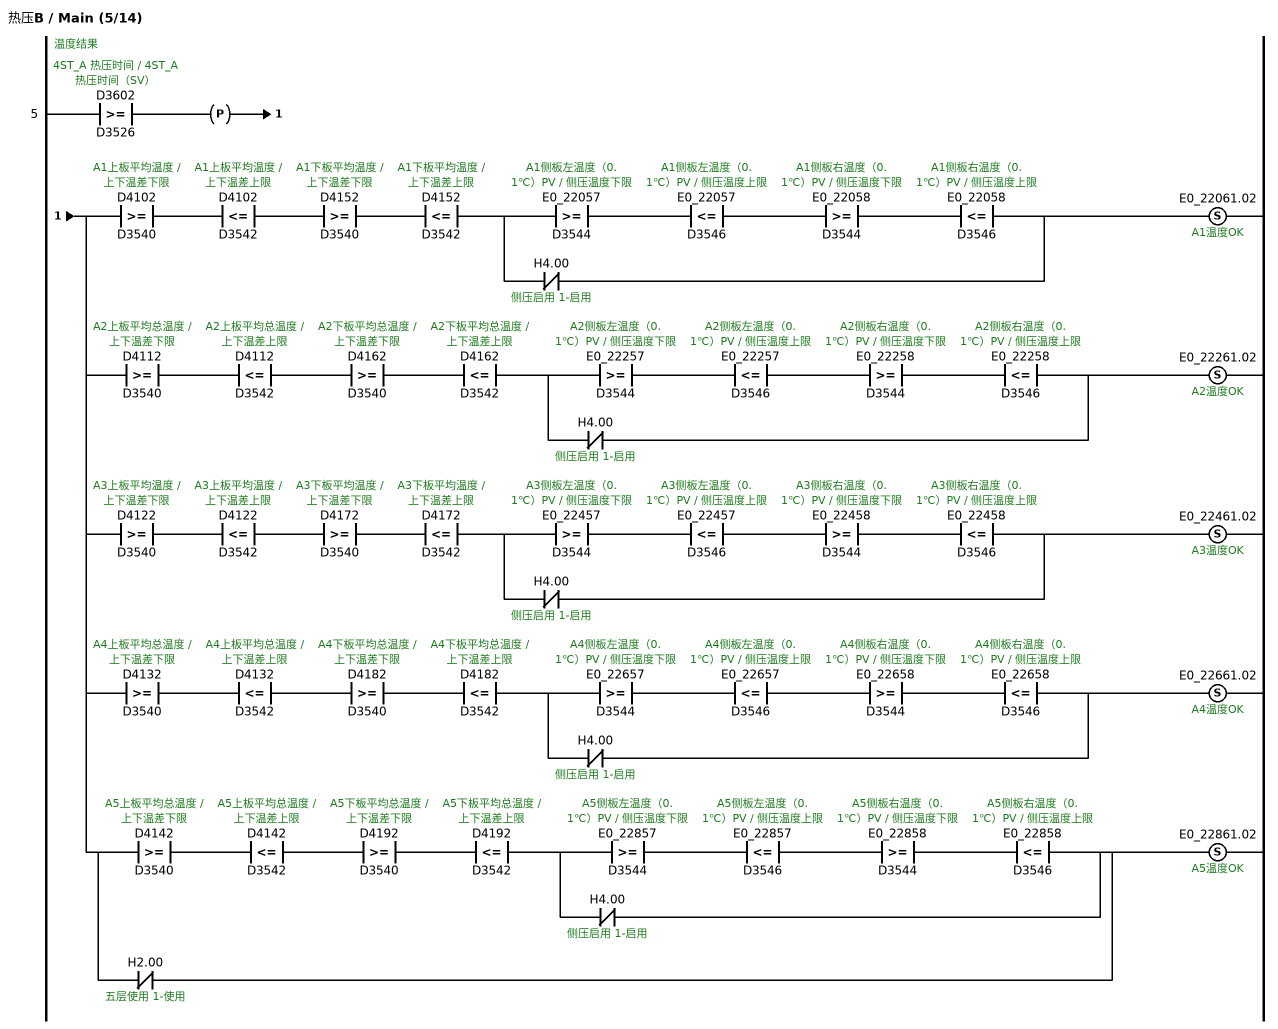
; [picture p168: 热压B / Main, rungs 5-5]
; rung 5: 温度结果
LD>=(325) D3602 D3526  ; 4ST_A 热压时间, 4ST_A 热压时间（SV）
UP(521)
OUT TR0
AND>=(325) D4102 D3540  ; A1上板平均温度, 上下温差下限
AND<=(315) D4102 D3542  ; A1上板平均温度, 上下温差上限
AND>=(325) D4152 D3540  ; A1下板平均温度, 上下温差下限
AND<=(315) D4152 D3542  ; A1下板平均温度, 上下温差上限
LD>=(325) E0_22057 D3544  ; A1侧板左温度（0.1℃）PV, 侧压温度下限
AND<=(315) E0_22057 D3546  ; A1侧板左温度（0.1℃）PV, 侧压温度上限
AND>=(325) E0_22058 D3544  ; A1侧板右温度（0.1℃）PV, 侧压温度下限
AND<=(315) E0_22058 D3546  ; A1侧板右温度（0.1℃）PV, 侧压温度上限
ORNOT H4.00  ; 侧压启用 1-启用
ANDLD
SET E0_22061.02  ; A1温度OK
LD TR0
AND>=(325) D4112 D3540  ; A2上板平均总温度, 上下温差下限
AND<=(315) D4112 D3542  ; A2上板平均总温度, 上下温差上限
AND>=(325) D4162 D3540  ; A2下板平均总温度, 上下温差下限
AND<=(315) D4162 D3542  ; A2下板平均总温度, 上下温差上限
LD>=(325) E0_22257 D3544  ; A2侧板左温度（0.1℃）PV, 侧压温度下限
AND<=(315) E0_22257 D3546  ; A2侧板左温度（0.1℃）PV, 侧压温度上限
AND>=(325) E0_22258 D3544  ; A2侧板右温度（0.1℃）PV, 侧压温度下限
AND<=(315) E0_22258 D3546  ; A2侧板右温度（0.1℃）PV, 侧压温度上限
ORNOT H4.00  ; 侧压启用 1-启用
ANDLD
SET E0_22261.02  ; A2温度OK
LD TR0
AND>=(325) D4122 D3540  ; A3上板平均温度, 上下温差下限
AND<=(315) D4122 D3542  ; A3上板平均温度, 上下温差上限
AND>=(325) D4172 D3540  ; A3下板平均温度, 上下温差下限
AND<=(315) D4172 D3542  ; A3下板平均温度, 上下温差上限
LD>=(325) E0_22457 D3544  ; A3侧板左温度（0.1℃）PV, 侧压温度下限
AND<=(315) E0_22457 D3546  ; A3侧板左温度（0.1℃）PV, 侧压温度上限
AND>=(325) E0_22458 D3544  ; A3侧板右温度（0.1℃）PV, 侧压温度下限
AND<=(315) E0_22458 D3546  ; A3侧板右温度（0.1℃）PV, 侧压温度上限
ORNOT H4.00  ; 侧压启用 1-启用
ANDLD
SET E0_22461.02  ; A3温度OK
LD TR0
AND>=(325) D4132 D3540  ; A4上板平均总温度, 上下温差下限
AND<=(315) D4132 D3542  ; A4上板平均总温度, 上下温差上限
AND>=(325) D4182 D3540  ; A4下板平均总温度, 上下温差下限
AND<=(315) D4182 D3542  ; A4下板平均总温度, 上下温差上限
LD>=(325) E0_22657 D3544  ; A4侧板左温度（0.1℃）PV, 侧压温度下限
AND<=(315) E0_22657 D3546  ; A4侧板左温度（0.1℃）PV, 侧压温度上限
AND>=(325) E0_22658 D3544  ; A4侧板右温度（0.1℃）PV, 侧压温度下限
AND<=(315) E0_22658 D3546  ; A4侧板右温度（0.1℃）PV, 侧压温度上限
ORNOT H4.00  ; 侧压启用 1-启用
ANDLD
SET E0_22661.02  ; A4温度OK
LD TR0
LD>=(325) D4142 D3540  ; A5上板平均总温度, 上下温差下限
AND<=(315) D4142 D3542  ; A5上板平均总温度, 上下温差上限
AND>=(325) D4192 D3540  ; A5下板平均总温度, 上下温差下限
AND<=(315) D4192 D3542  ; A5下板平均总温度, 上下温差上限
LD>=(325) E0_22857 D3544  ; A5侧板左温度（0.1℃）PV, 侧压温度下限
AND<=(315) E0_22857 D3546  ; A5侧板左温度（0.1℃）PV, 侧压温度上限
AND>=(325) E0_22858 D3544  ; A5侧板右温度（0.1℃）PV, 侧压温度下限
AND<=(315) E0_22858 D3546  ; A5侧板右温度（0.1℃）PV, 侧压温度上限
ORNOT H4.00  ; 侧压启用 1-启用
ANDLD
ORNOT H2.00  ; 五层使用 1-使用
ANDLD
SET E0_22861.02  ; A5温度OK

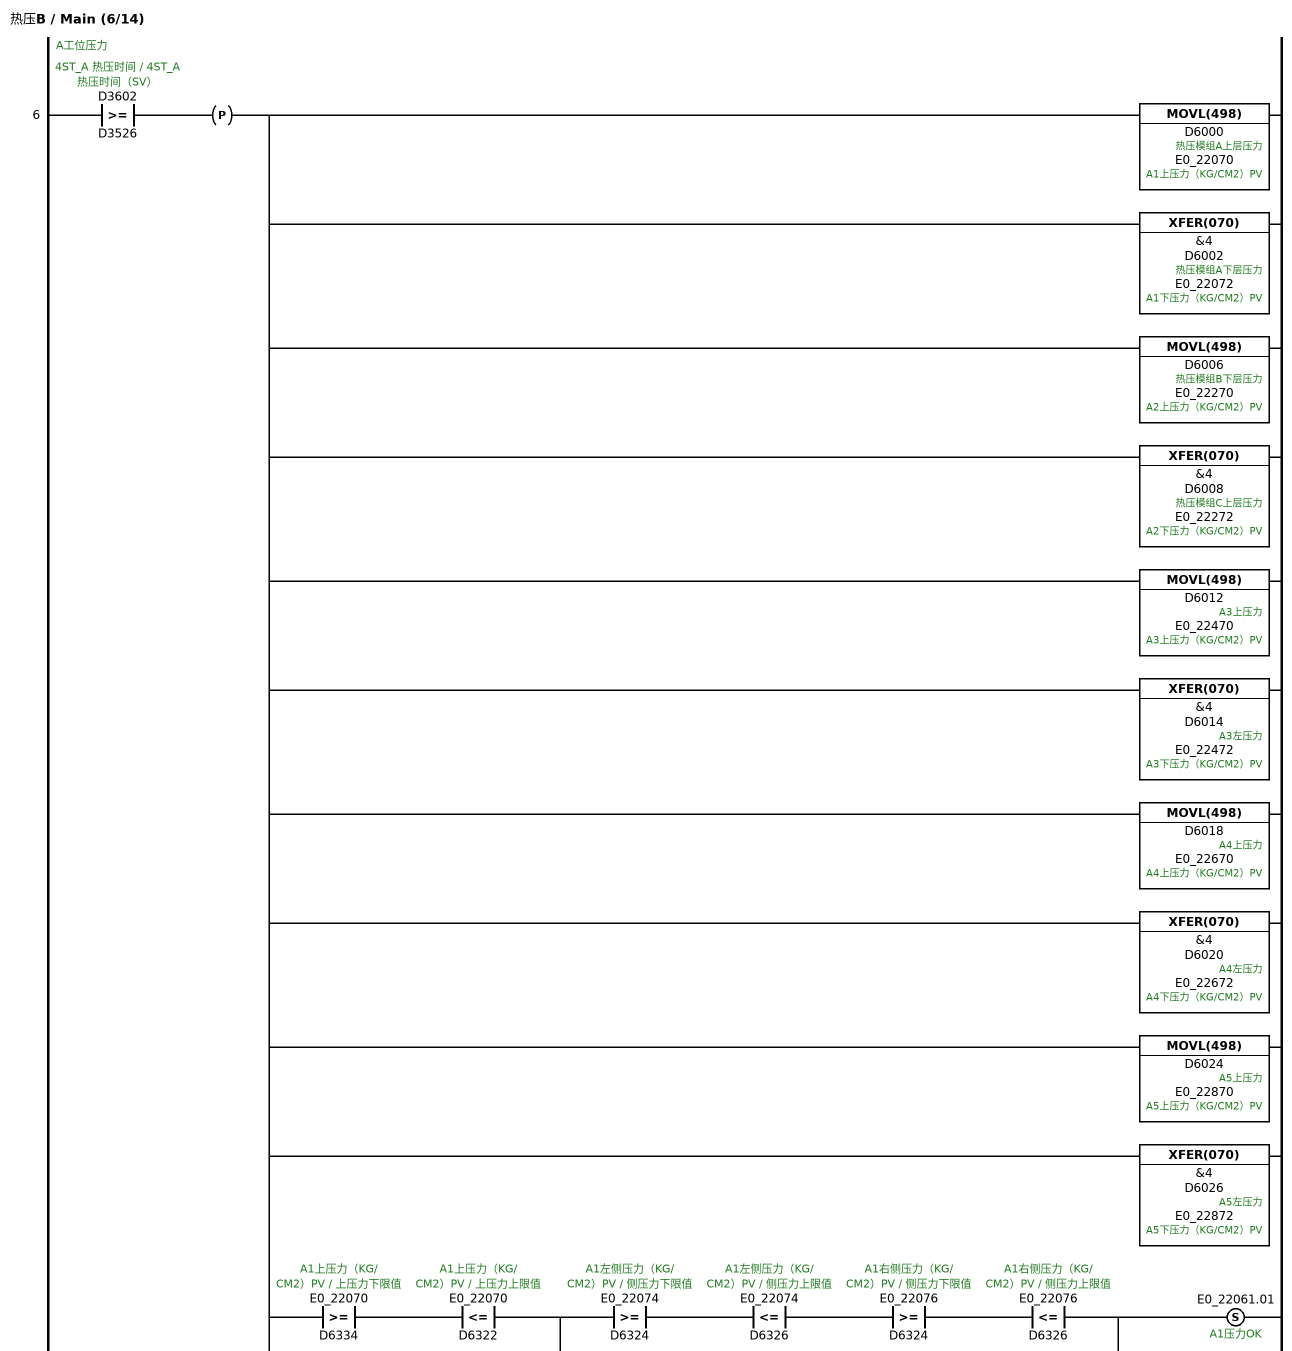

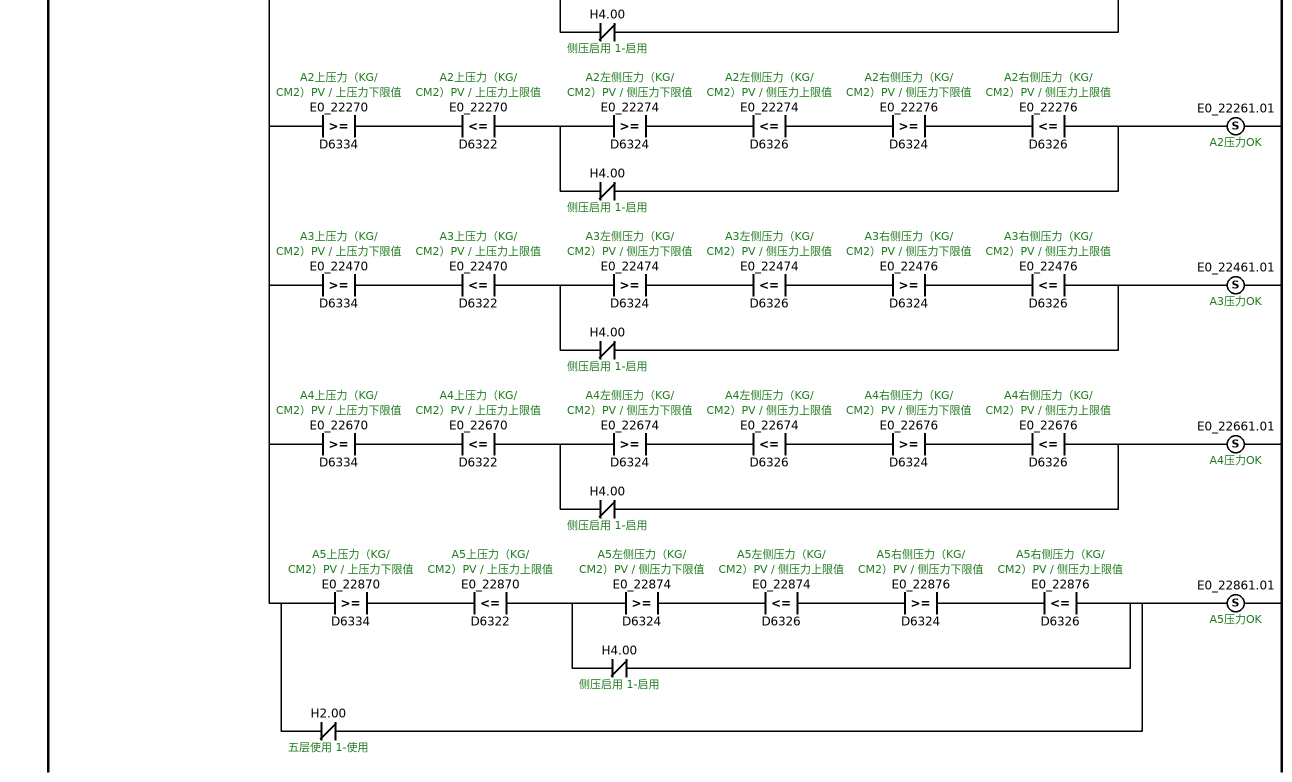
; rung 6: A工位压力
LD>=(325) D3602 D3526  ; 4ST_A 热压时间, 4ST_A 热压时间（SV）
UP(521)
OUT TR0
MOVL(498) D6000 E0_22070  ; 热压模组A上层压力, A1上压力（KG/CM2）PV
XFER(070) &4 D6002 E0_22072  ; 热压模组A下层压力, A1下压力（KG/CM2）PV
MOVL(498) D6006 E0_22270  ; 热压模组B下层压力, A2上压力（KG/CM2）PV
XFER(070) &4 D6008 E0_22272  ; 热压模组C上层压力, A2下压力（KG/CM2）PV
MOVL(498) D6012 E0_22470  ; A3上压力, A3上压力（KG/CM2）PV
XFER(070) &4 D6014 E0_22472  ; A3左压力, A3下压力（KG/CM2）PV
MOVL(498) D6018 E0_22670  ; A4上压力, A4上压力（KG/CM2）PV
XFER(070) &4 D6020 E0_22672  ; A4左压力, A4下压力（KG/CM2）PV
MOVL(498) D6024 E0_22870  ; A5上压力, A5上压力（KG/CM2）PV
XFER(070) &4 D6026 E0_22872  ; A5左压力, A5下压力（KG/CM2）PV
AND>=L(326) E0_22070 D6334  ; A1上压力（KG/CM2）PV, 上压力下限值
AND<=L(316) E0_22070 D6322  ; A1上压力（KG/CM2）PV, 上压力上限值
LD>=L(326) E0_22074 D6324  ; A1左侧压力（KG/CM2）PV, 侧压力下限值
AND<=L(316) E0_22074 D6326  ; A1左侧压力（KG/CM2）PV, 侧压力上限值
AND>=L(326) E0_22076 D6324  ; A1右侧压力（KG/CM2）PV, 侧压力下限值
AND<=L(316) E0_22076 D6326  ; A1右侧压力（KG/CM2）PV, 侧压力上限值
ORNOT H4.00  ; 侧压启用 1-启用
ANDLD
SET E0_22061.01  ; A1压力OK
LD TR0
AND>=L(326) E0_22270 D6334  ; A2上压力（KG/CM2）PV, 上压力下限值
AND<=L(316) E0_22270 D6322  ; A2上压力（KG/CM2）PV, 上压力上限值
LD>=L(326) E0_22274 D6324  ; A2左侧压力（KG/CM2）PV, 侧压力下限值
AND<=L(316) E0_22274 D6326  ; A2左侧压力（KG/CM2）PV, 侧压力上限值
AND>=L(326) E0_22276 D6324  ; A2右侧压力（KG/CM2）PV, 侧压力下限值
AND<=L(316) E0_22276 D6326  ; A2右侧压力（KG/CM2）PV, 侧压力上限值
ORNOT H4.00  ; 侧压启用 1-启用
ANDLD
SET E0_22261.01  ; A2压力OK
LD TR0
AND>=L(326) E0_22470 D6334  ; A3上压力（KG/CM2）PV, 上压力下限值
AND<=L(316) E0_22470 D6322  ; A3上压力（KG/CM2）PV, 上压力上限值
LD>=L(326) E0_22474 D6324  ; A3左侧压力（KG/CM2）PV, 侧压力下限值
AND<=L(316) E0_22474 D6326  ; A3左侧压力（KG/CM2）PV, 侧压力上限值
AND>=L(326) E0_22476 D6324  ; A3右侧压力（KG/CM2）PV, 侧压力下限值
AND<=L(316) E0_22476 D6326  ; A3右侧压力（KG/CM2）PV, 侧压力上限值
ORNOT H4.00  ; 侧压启用 1-启用
ANDLD
SET E0_22461.01  ; A3压力OK
LD TR0
AND>=L(326) E0_22670 D6334  ; A4上压力（KG/CM2）PV, 上压力下限值
AND<=L(316) E0_22670 D6322  ; A4上压力（KG/CM2）PV, 上压力上限值
LD>=L(326) E0_22674 D6324  ; A4左侧压力（KG/CM2）PV, 侧压力下限值
AND<=L(316) E0_22674 D6326  ; A4左侧压力（KG/CM2）PV, 侧压力上限值
AND>=L(326) E0_22676 D6324  ; A4右侧压力（KG/CM2）PV, 侧压力下限值
AND<=L(316) E0_22676 D6326  ; A4右侧压力（KG/CM2）PV, 侧压力上限值
ORNOT H4.00  ; 侧压启用 1-启用
ANDLD
SET E0_22661.01  ; A4压力OK
LD TR0
LD>=L(326) E0_22870 D6334  ; A5上压力（KG/CM2）PV, 上压力下限值
AND<=L(316) E0_22870 D6322  ; A5上压力（KG/CM2）PV, 上压力上限值
LD>=L(326) E0_22874 D6324  ; A5左侧压力（KG/CM2）PV, 侧压力下限值
AND<=L(316) E0_22874 D6326  ; A5左侧压力（KG/CM2）PV, 侧压力上限值
AND>=L(326) E0_22876 D6324  ; A5右侧压力（KG/CM2）PV, 侧压力下限值
AND<=L(316) E0_22876 D6326  ; A5右侧压力（KG/CM2）PV, 侧压力上限值
ORNOT H4.00  ; 侧压启用 1-启用
ANDLD
ORNOT H2.00  ; 五层使用 1-使用
ANDLD
SET E0_22861.01  ; A5压力OK

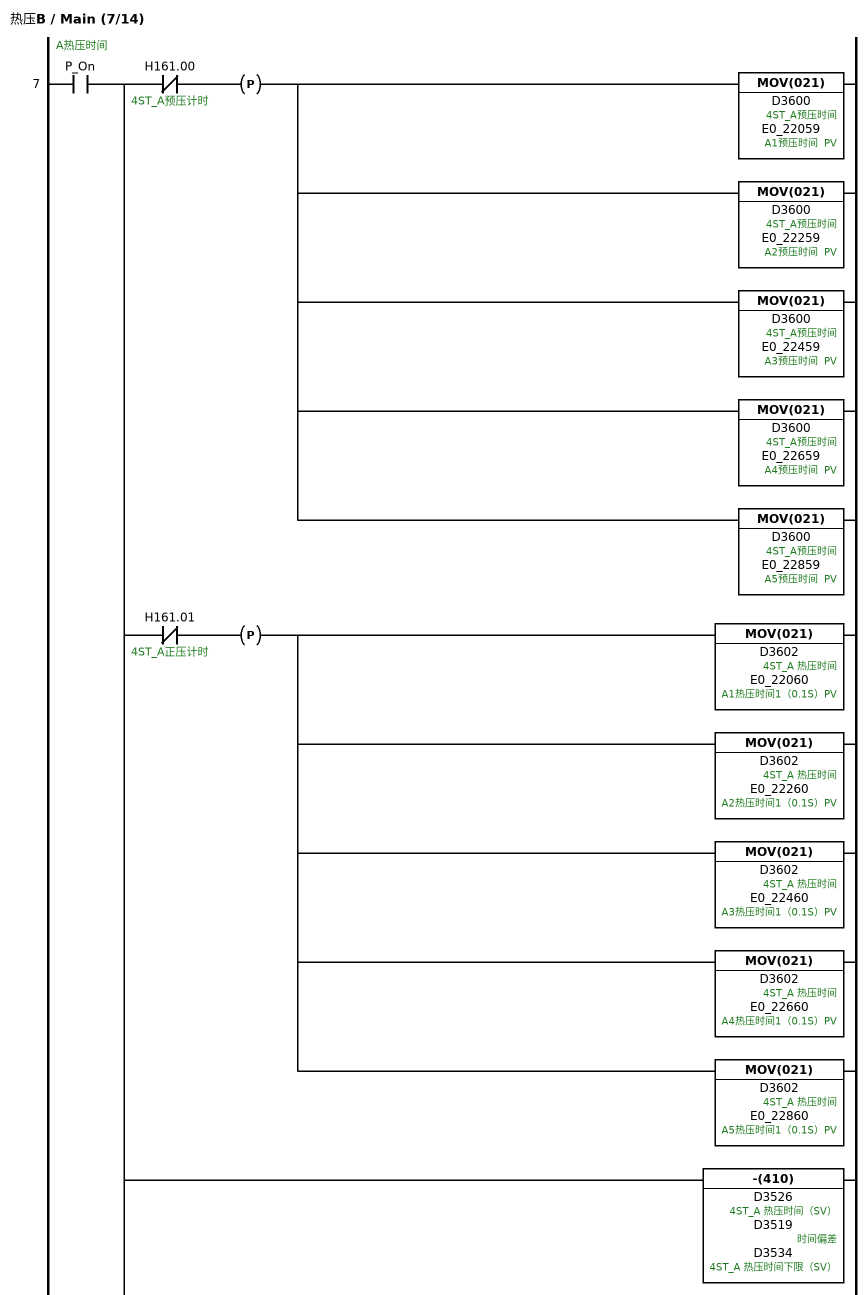

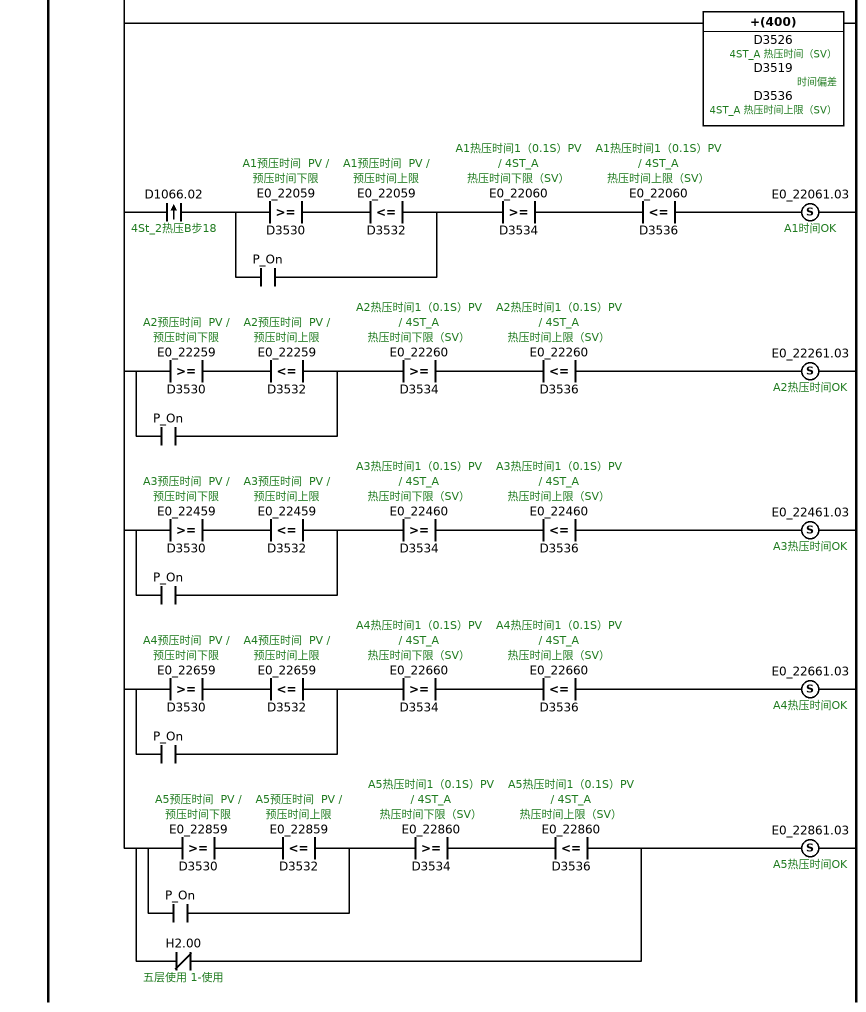
; rung 7: A热压时间
LD P_On
OUT TR0
ANDNOT H161.00  ; 4ST_A预压计时
UP(521)
MOV(021) D3600 E0_22059  ; 4ST_A预压时间, A1预压时间  PV
MOV(021) D3600 E0_22259  ; 4ST_A预压时间, A2预压时间  PV
MOV(021) D3600 E0_22459  ; 4ST_A预压时间, A3预压时间  PV
MOV(021) D3600 E0_22659  ; 4ST_A预压时间, A4预压时间  PV
MOV(021) D3600 E0_22859  ; 4ST_A预压时间, A5预压时间  PV
LD TR0
ANDNOT H161.01  ; 4ST_A正压计时
UP(521)
MOV(021) D3602 E0_22060  ; 4ST_A 热压时间, A1热压时间1（0.1S）PV
MOV(021) D3602 E0_22260  ; 4ST_A 热压时间, A2热压时间1（0.1S）PV
MOV(021) D3602 E0_22460  ; 4ST_A 热压时间, A3热压时间1（0.1S）PV
MOV(021) D3602 E0_22660  ; 4ST_A 热压时间, A4热压时间1（0.1S）PV
MOV(021) D3602 E0_22860  ; 4ST_A 热压时间, A5热压时间1（0.1S）PV
LD TR0
-(410) D3526 D3519 D3534  ; 4ST_A 热压时间（SV）, 时间偏差, 4ST_A 热压时间下限（SV）
+(400) D3526 D3519 D3536  ; 4ST_A 热压时间（SV）, 时间偏差, 4ST_A 热压时间上限（SV）
@AND D1066.02  ; 4St_2热压B步18
LD>=(325) E0_22059 D3530  ; A1预压时间  PV, 预压时间下限
AND<=(315) E0_22059 D3532  ; A1预压时间  PV, 预压时间上限
OR P_On
ANDLD
AND>=(325) E0_22060 D3534  ; A1热压时间1（0.1S）PV, 4ST_A 热压时间下限（SV）
AND<=(315) E0_22060 D3536  ; A1热压时间1（0.1S）PV, 4ST_A 热压时间上限（SV）
SET E0_22061.03  ; A1时间OK
LD TR0
LD>=(325) E0_22259 D3530  ; A2预压时间  PV, 预压时间下限
AND<=(315) E0_22259 D3532  ; A2预压时间  PV, 预压时间上限
OR P_On
ANDLD
AND>=(325) E0_22260 D3534  ; A2热压时间1（0.1S）PV, 4ST_A 热压时间下限（SV）
AND<=(315) E0_22260 D3536  ; A2热压时间1（0.1S）PV, 4ST_A 热压时间上限（SV）
SET E0_22261.03  ; A2热压时间OK
LD TR0
LD>=(325) E0_22459 D3530  ; A3预压时间  PV, 预压时间下限
AND<=(315) E0_22459 D3532  ; A3预压时间  PV, 预压时间上限
OR P_On
ANDLD
AND>=(325) E0_22460 D3534  ; A3热压时间1（0.1S）PV, 4ST_A 热压时间下限（SV）
AND<=(315) E0_22460 D3536  ; A3热压时间1（0.1S）PV, 4ST_A 热压时间上限（SV）
SET E0_22461.03  ; A3热压时间OK
LD TR0
LD>=(325) E0_22659 D3530  ; A4预压时间  PV, 预压时间下限
AND<=(315) E0_22659 D3532  ; A4预压时间  PV, 预压时间上限
OR P_On
ANDLD
AND>=(325) E0_22660 D3534  ; A4热压时间1（0.1S）PV, 4ST_A 热压时间下限（SV）
AND<=(315) E0_22660 D3536  ; A4热压时间1（0.1S）PV, 4ST_A 热压时间上限（SV）
SET E0_22661.03  ; A4热压时间OK
LD TR0
LD>=(325) E0_22859 D3530  ; A5预压时间  PV, 预压时间下限
AND<=(315) E0_22859 D3532  ; A5预压时间  PV, 预压时间上限
OR P_On
AND>=(325) E0_22860 D3534  ; A5热压时间1（0.1S）PV, 4ST_A 热压时间下限（SV）
AND<=(315) E0_22860 D3536  ; A5热压时间1（0.1S）PV, 4ST_A 热压时间上限（SV）
ORNOT H2.00  ; 五层使用 1-使用
ANDLD
SET E0_22861.03  ; A5热压时间OK

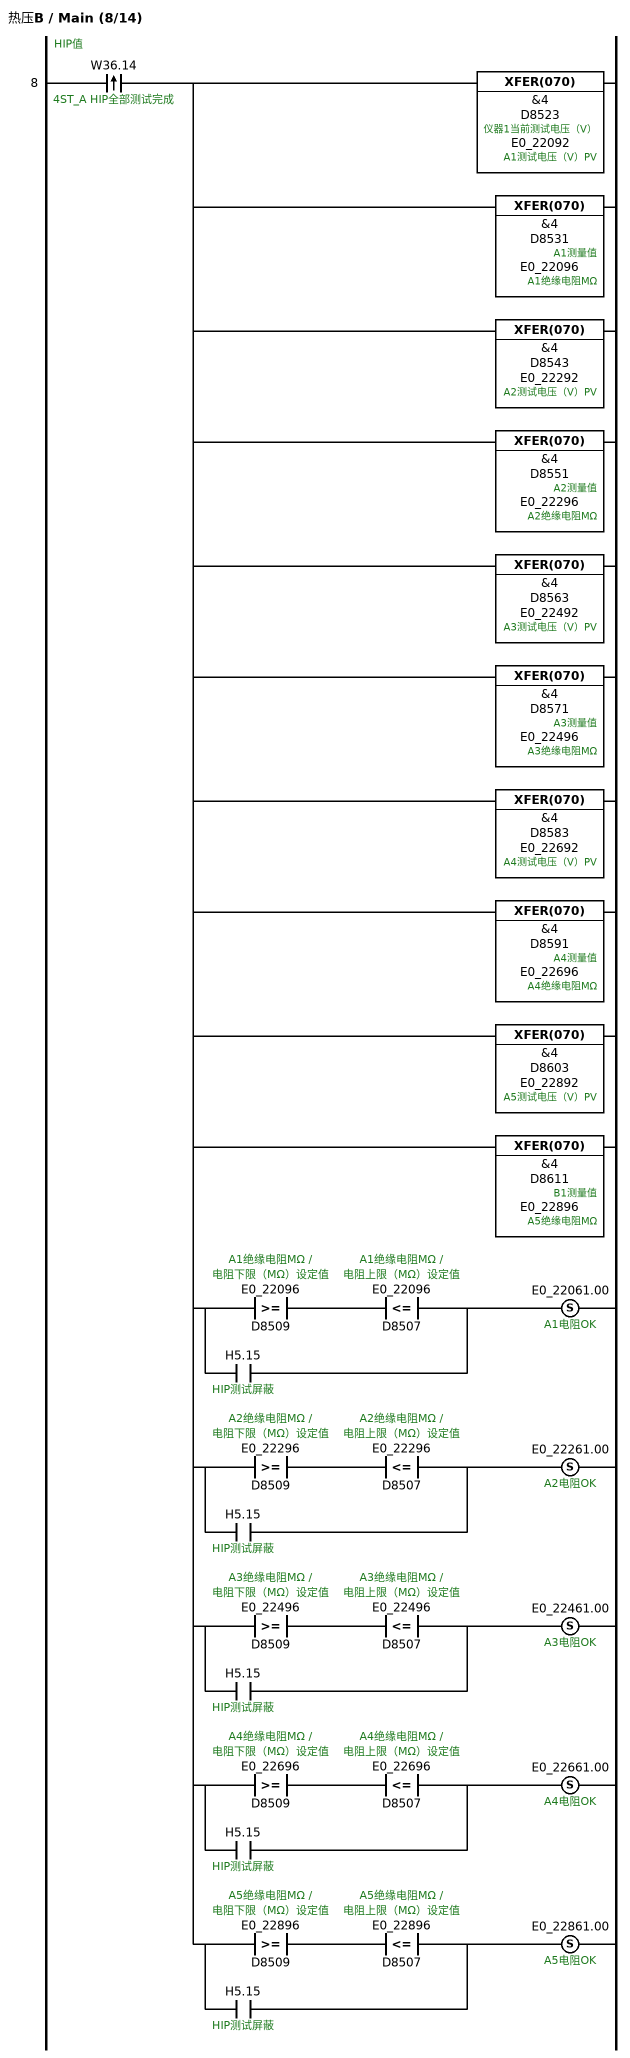
; rung 8: HIP值
@LD W36.14  ; 4ST_A HIP全部测试完成
OUT TR0
XFER(070) &4 D8523 E0_22092  ; 仪器1当前测试电压（V）, A1测试电压（V）PV
XFER(070) &4 D8531 E0_22096  ; A1测量值, A1绝缘电阻MΩ
XFER(070) &4 D8543 E0_22292  ; A2测试电压（V）PV
XFER(070) &4 D8551 E0_22296  ; A2测量值, A2绝缘电阻MΩ
XFER(070) &4 D8563 E0_22492  ; A3测试电压（V）PV
XFER(070) &4 D8571 E0_22496  ; A3测量值, A3绝缘电阻MΩ
XFER(070) &4 D8583 E0_22692  ; A4测试电压（V）PV
XFER(070) &4 D8591 E0_22696  ; A4测量值, A4绝缘电阻MΩ
XFER(070) &4 D8603 E0_22892  ; A5测试电压（V）PV
XFER(070) &4 D8611 E0_22896  ; B1测量值, A5绝缘电阻MΩ
LD>=F(334) E0_22096 D8509  ; A1绝缘电阻MΩ, 电阻下限（MΩ）设定值
AND<=F(332) E0_22096 D8507  ; A1绝缘电阻MΩ, 电阻上限（MΩ）设定值
OR H5.15  ; HIP测试屏蔽
ANDLD
SET E0_22061.00  ; A1电阻OK
LD TR0
LD>=F(334) E0_22296 D8509  ; A2绝缘电阻MΩ, 电阻下限（MΩ）设定值
AND<=F(332) E0_22296 D8507  ; A2绝缘电阻MΩ, 电阻上限（MΩ）设定值
OR H5.15  ; HIP测试屏蔽
ANDLD
SET E0_22261.00  ; A2电阻OK
LD TR0
LD>=F(334) E0_22496 D8509  ; A3绝缘电阻MΩ, 电阻下限（MΩ）设定值
AND<=F(332) E0_22496 D8507  ; A3绝缘电阻MΩ, 电阻上限（MΩ）设定值
OR H5.15  ; HIP测试屏蔽
ANDLD
SET E0_22461.00  ; A3电阻OK
LD TR0
LD>=F(334) E0_22696 D8509  ; A4绝缘电阻MΩ, 电阻下限（MΩ）设定值
AND<=F(332) E0_22696 D8507  ; A4绝缘电阻MΩ, 电阻上限（MΩ）设定值
OR H5.15  ; HIP测试屏蔽
ANDLD
SET E0_22661.00  ; A4电阻OK
LD TR0
LD>=F(334) E0_22896 D8509  ; A5绝缘电阻MΩ, 电阻下限（MΩ）设定值
AND<=F(332) E0_22896 D8507  ; A5绝缘电阻MΩ, 电阻上限（MΩ）设定值
OR H5.15  ; HIP测试屏蔽
ANDLD
SET E0_22861.00  ; A5电阻OK

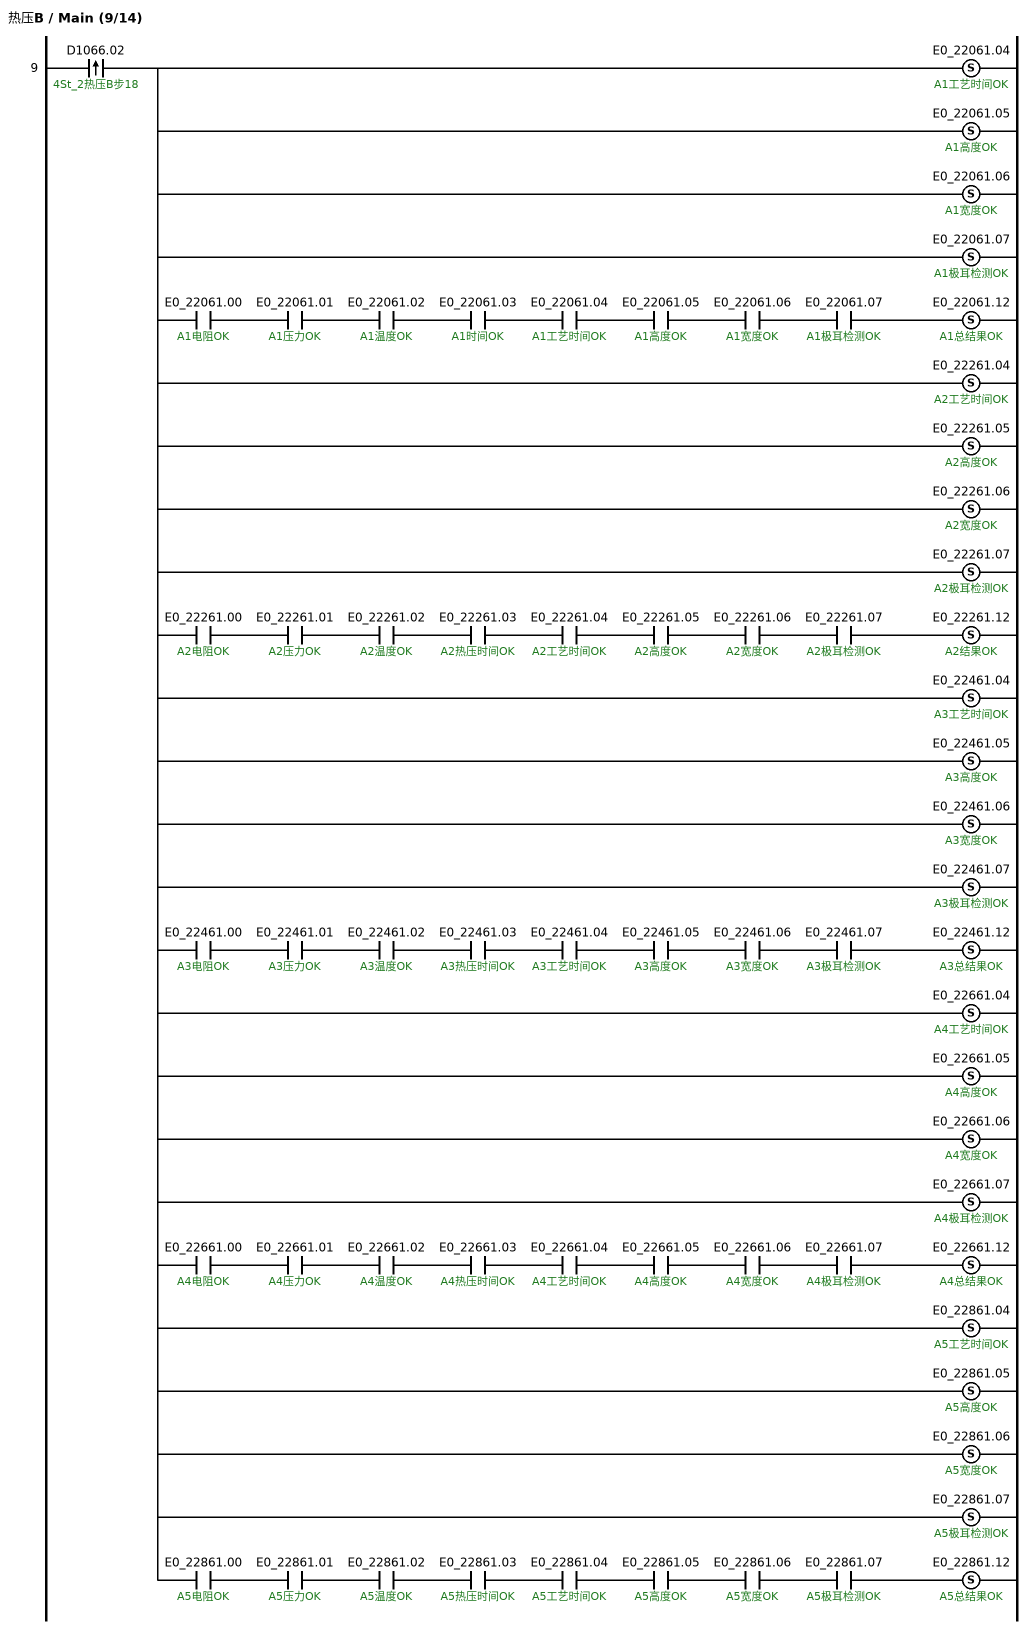
; rung 9
@LD D1066.02  ; 4St_2热压B步18
OUT TR0
SET E0_22061.04  ; A1工艺时间OK
SET E0_22061.05  ; A1高度OK
SET E0_22061.06  ; A1宽度OK
SET E0_22061.07  ; A1极耳检测OK
AND E0_22061.00  ; A1电阻OK
AND E0_22061.01  ; A1压力OK
AND E0_22061.02  ; A1温度OK
AND E0_22061.03  ; A1时间OK
AND E0_22061.04  ; A1工艺时间OK
AND E0_22061.05  ; A1高度OK
AND E0_22061.06  ; A1宽度OK
AND E0_22061.07  ; A1极耳检测OK
SET E0_22061.12  ; A1总结果OK
LD TR0
SET E0_22261.04  ; A2工艺时间OK
SET E0_22261.05  ; A2高度OK
SET E0_22261.06  ; A2宽度OK
SET E0_22261.07  ; A2极耳检测OK
AND E0_22261.00  ; A2电阻OK
AND E0_22261.01  ; A2压力OK
AND E0_22261.02  ; A2温度OK
AND E0_22261.03  ; A2热压时间OK
AND E0_22261.04  ; A2工艺时间OK
AND E0_22261.05  ; A2高度OK
AND E0_22261.06  ; A2宽度OK
AND E0_22261.07  ; A2极耳检测OK
SET E0_22261.12  ; A2结果OK
LD TR0
SET E0_22461.04  ; A3工艺时间OK
SET E0_22461.05  ; A3高度OK
SET E0_22461.06  ; A3宽度OK
SET E0_22461.07  ; A3极耳检测OK
AND E0_22461.00  ; A3电阻OK
AND E0_22461.01  ; A3压力OK
AND E0_22461.02  ; A3温度OK
AND E0_22461.03  ; A3热压时间OK
AND E0_22461.04  ; A3工艺时间OK
AND E0_22461.05  ; A3高度OK
AND E0_22461.06  ; A3宽度OK
AND E0_22461.07  ; A3极耳检测OK
SET E0_22461.12  ; A3总结果OK
LD TR0
SET E0_22661.04  ; A4工艺时间OK
SET E0_22661.05  ; A4高度OK
SET E0_22661.06  ; A4宽度OK
SET E0_22661.07  ; A4极耳检测OK
AND E0_22661.00  ; A4电阻OK
AND E0_22661.01  ; A4压力OK
AND E0_22661.02  ; A4温度OK
AND E0_22661.03  ; A4热压时间OK
AND E0_22661.04  ; A4工艺时间OK
AND E0_22661.05  ; A4高度OK
AND E0_22661.06  ; A4宽度OK
AND E0_22661.07  ; A4极耳检测OK
SET E0_22661.12  ; A4总结果OK
LD TR0
SET E0_22861.04  ; A5工艺时间OK
SET E0_22861.05  ; A5高度OK
SET E0_22861.06  ; A5宽度OK
SET E0_22861.07  ; A5极耳检测OK
AND E0_22861.00  ; A5电阻OK
AND E0_22861.01  ; A5压力OK
AND E0_22861.02  ; A5温度OK
AND E0_22861.03  ; A5热压时间OK
AND E0_22861.04  ; A5工艺时间OK
AND E0_22861.05  ; A5高度OK
AND E0_22861.06  ; A5宽度OK
AND E0_22861.07  ; A5极耳检测OK
SET E0_22861.12  ; A5总结果OK

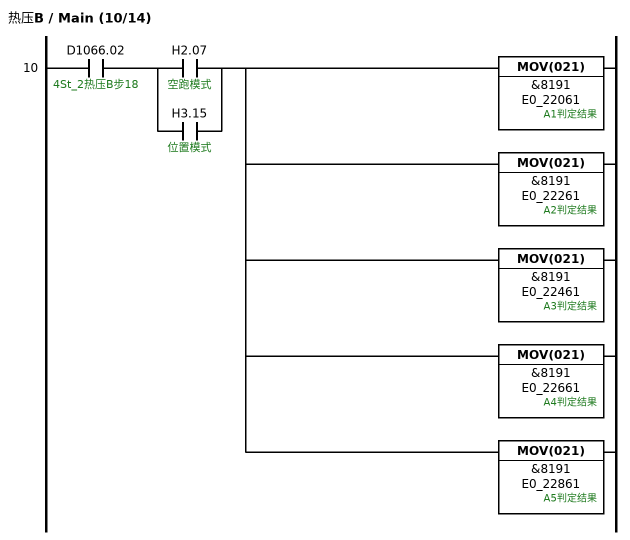
; rung 10
LD D1066.02  ; 4St_2热压B步18
LD H2.07  ; 空跑模式
OR H3.15  ; 位置模式
ANDLD
MOV(021) &8191 E0_22061  ; A1判定结果
MOV(021) &8191 E0_22261  ; A2判定结果
MOV(021) &8191 E0_22461  ; A3判定结果
MOV(021) &8191 E0_22661  ; A4判定结果
MOV(021) &8191 E0_22861  ; A5判定结果

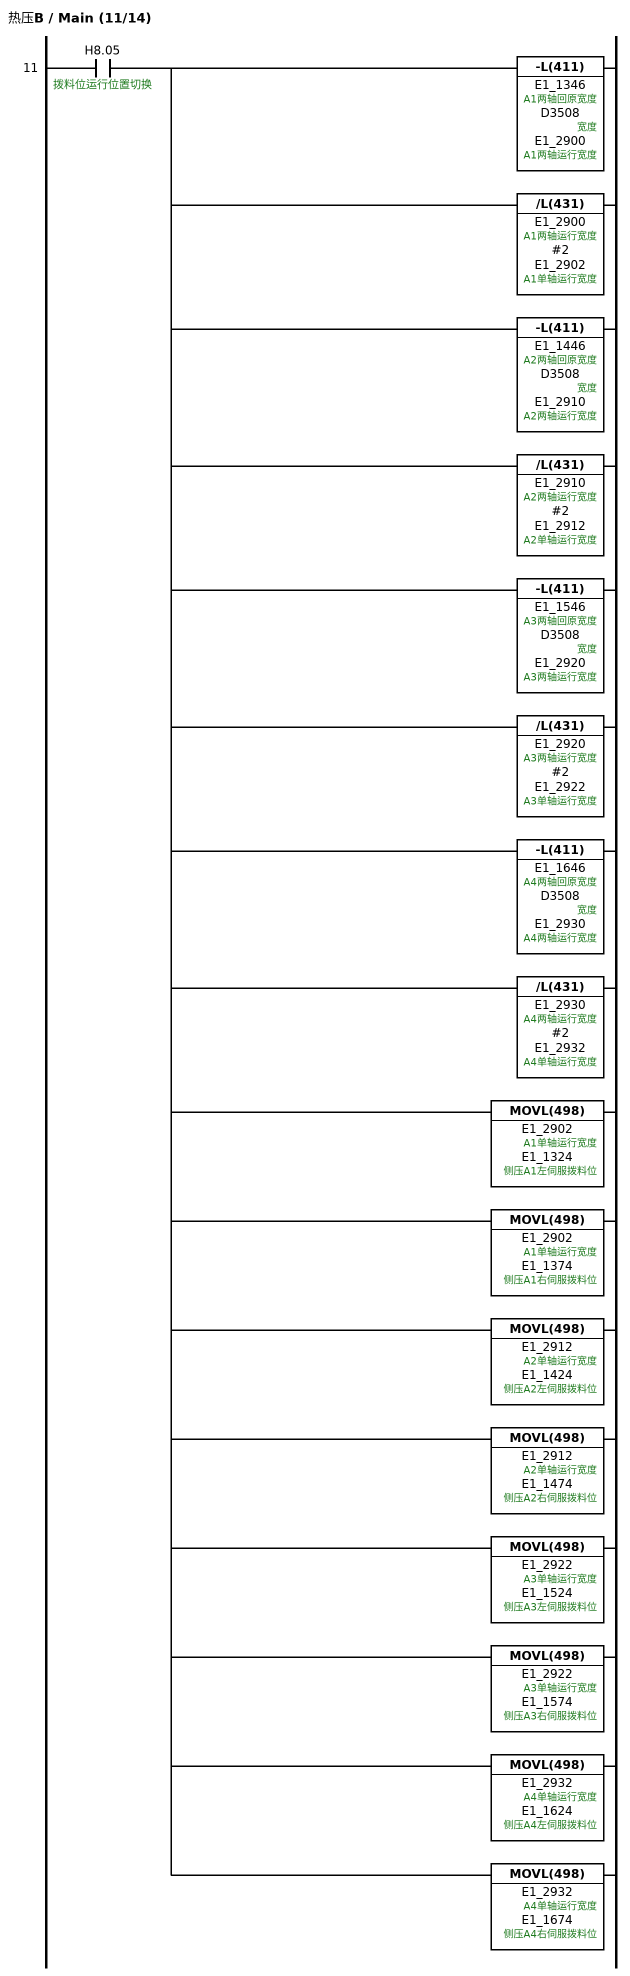
; rung 11
LD H8.05  ; 拨料位运行位置切换
-L(411) E1_1346 D3508 E1_2900  ; A1两轴回原宽度, 宽度, A1两轴运行宽度
/L(431) E1_2900 #2 E1_2902  ; A1两轴运行宽度, A1单轴运行宽度
-L(411) E1_1446 D3508 E1_2910  ; A2两轴回原宽度, 宽度, A2两轴运行宽度
/L(431) E1_2910 #2 E1_2912  ; A2两轴运行宽度, A2单轴运行宽度
-L(411) E1_1546 D3508 E1_2920  ; A3两轴回原宽度, 宽度, A3两轴运行宽度
/L(431) E1_2920 #2 E1_2922  ; A3两轴运行宽度, A3单轴运行宽度
-L(411) E1_1646 D3508 E1_2930  ; A4两轴回原宽度, 宽度, A4两轴运行宽度
/L(431) E1_2930 #2 E1_2932  ; A4两轴运行宽度, A4单轴运行宽度
MOVL(498) E1_2902 E1_1324  ; A1单轴运行宽度, 侧压A1左伺服拨料位
MOVL(498) E1_2902 E1_1374  ; A1单轴运行宽度, 侧压A1右伺服拨料位
MOVL(498) E1_2912 E1_1424  ; A2单轴运行宽度, 侧压A2左伺服拨料位
MOVL(498) E1_2912 E1_1474  ; A2单轴运行宽度, 侧压A2右伺服拨料位
MOVL(498) E1_2922 E1_1524  ; A3单轴运行宽度, 侧压A3左伺服拨料位
MOVL(498) E1_2922 E1_1574  ; A3单轴运行宽度, 侧压A3右伺服拨料位
MOVL(498) E1_2932 E1_1624  ; A4单轴运行宽度, 侧压A4左伺服拨料位
MOVL(498) E1_2932 E1_1674  ; A4单轴运行宽度, 侧压A4右伺服拨料位

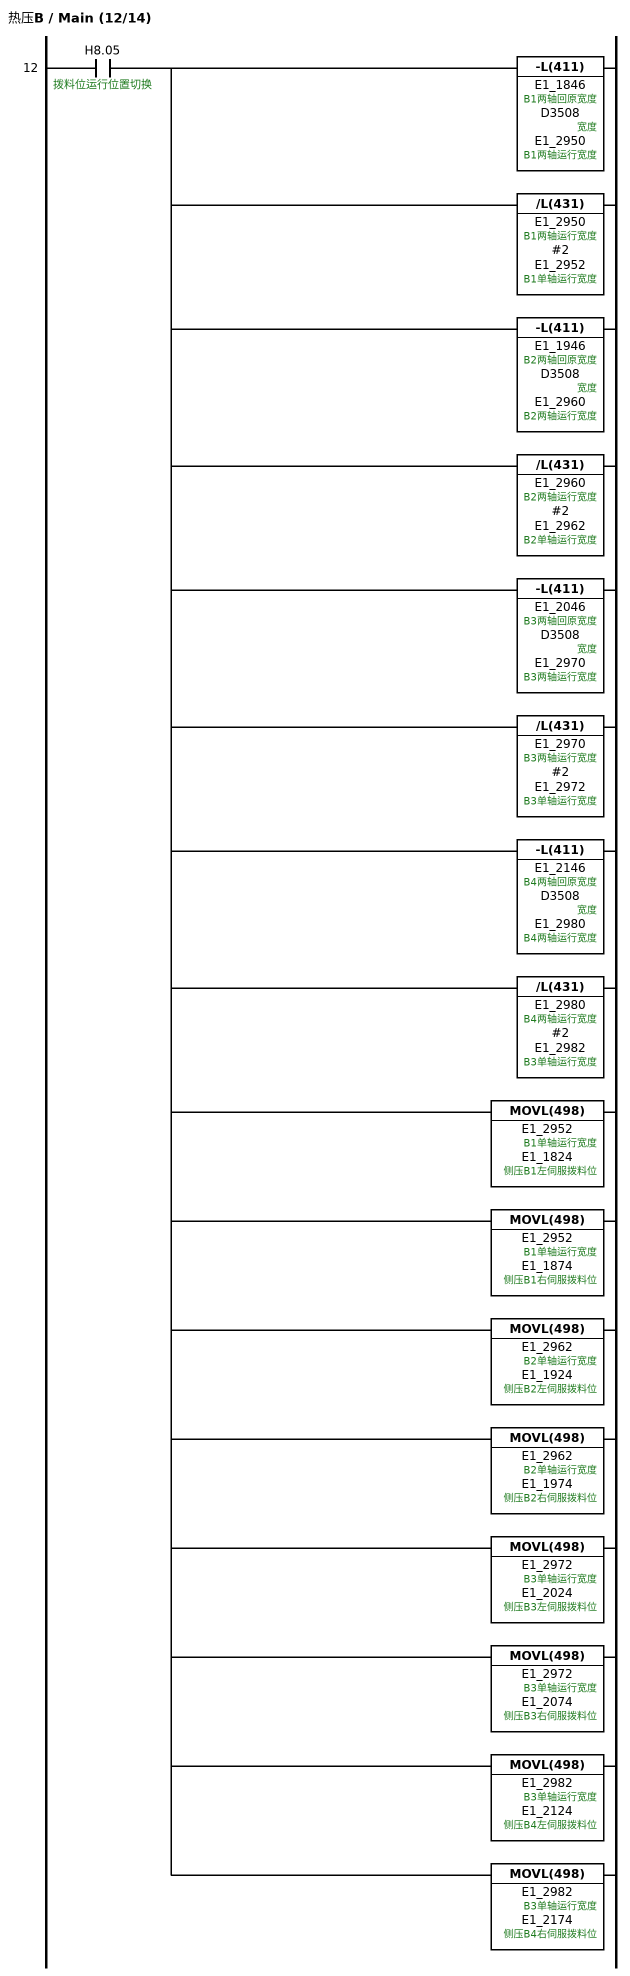
; rung 12
LD H8.05  ; 拨料位运行位置切换
-L(411) E1_1846 D3508 E1_2950  ; B1两轴回原宽度, 宽度, B1两轴运行宽度
/L(431) E1_2950 #2 E1_2952  ; B1两轴运行宽度, B1单轴运行宽度
-L(411) E1_1946 D3508 E1_2960  ; B2两轴回原宽度, 宽度, B2两轴运行宽度
/L(431) E1_2960 #2 E1_2962  ; B2两轴运行宽度, B2单轴运行宽度
-L(411) E1_2046 D3508 E1_2970  ; B3两轴回原宽度, 宽度, B3两轴运行宽度
/L(431) E1_2970 #2 E1_2972  ; B3两轴运行宽度, B3单轴运行宽度
-L(411) E1_2146 D3508 E1_2980  ; B4两轴回原宽度, 宽度, B4两轴运行宽度
/L(431) E1_2980 #2 E1_2982  ; B4两轴运行宽度, B3单轴运行宽度
MOVL(498) E1_2952 E1_1824  ; B1单轴运行宽度, 侧压B1左伺服拨料位
MOVL(498) E1_2952 E1_1874  ; B1单轴运行宽度, 侧压B1右伺服拨料位
MOVL(498) E1_2962 E1_1924  ; B2单轴运行宽度, 侧压B2左伺服拨料位
MOVL(498) E1_2962 E1_1974  ; B2单轴运行宽度, 侧压B2右伺服拨料位
MOVL(498) E1_2972 E1_2024  ; B3单轴运行宽度, 侧压B3左伺服拨料位
MOVL(498) E1_2972 E1_2074  ; B3单轴运行宽度, 侧压B3右伺服拨料位
MOVL(498) E1_2982 E1_2124  ; B3单轴运行宽度, 侧压B4左伺服拨料位
MOVL(498) E1_2982 E1_2174  ; B3单轴运行宽度, 侧压B4右伺服拨料位

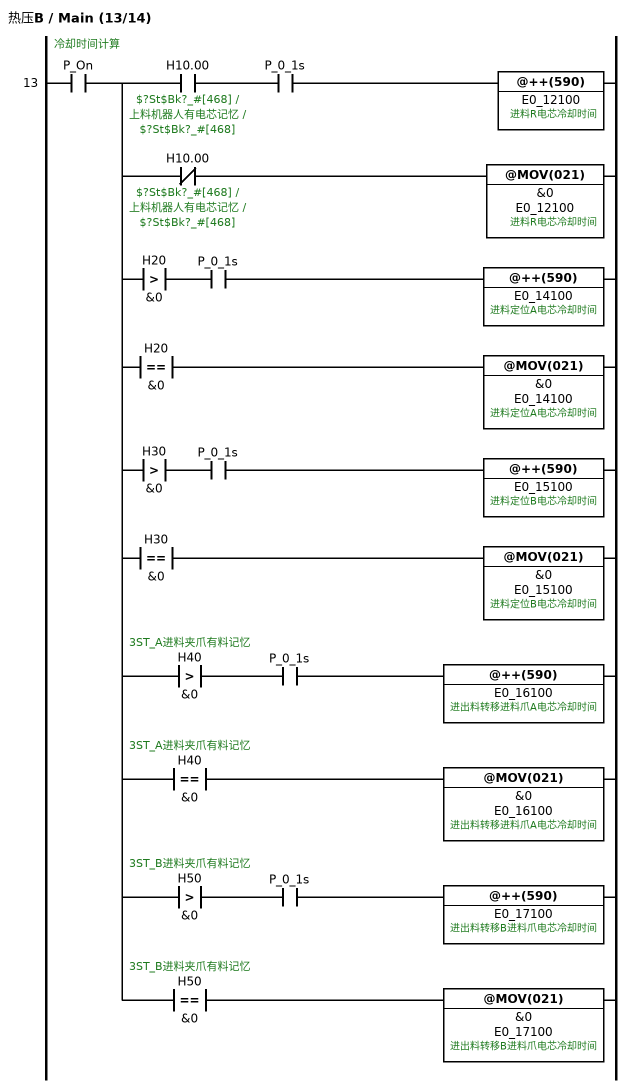
; rung 13: 冷却时间计算
LD P_On
OUT TR0
AND H10.00  ; $?St$Bk?_#[468] / 上料机器人有电芯记忆 / $?St$Bk?_#[468]
AND P_0_1s
@++(590) E0_12100  ; 进料R电芯冷却时间
LD TR0
ANDNOT H10.00  ; $?St$Bk?_#[468] / 上料机器人有电芯记忆 / $?St$Bk?_#[468]
@MOV(021) &0 E0_12100  ; 进料R电芯冷却时间
LD TR0
AND>(320) H20 &0
AND P_0_1s
@++(590) E0_14100  ; 进料定位A电芯冷却时间
LD TR0
AND=(300) H20 &0
@MOV(021) &0 E0_14100  ; 进料定位A电芯冷却时间
LD TR0
AND>(320) H30 &0
AND P_0_1s
@++(590) E0_15100  ; 进料定位B电芯冷却时间
LD TR0
AND=(300) H30 &0
@MOV(021) &0 E0_15100  ; 进料定位B电芯冷却时间
LD TR0
AND>(320) H40 &0  ; 3ST_A进料夹爪有料记忆
AND P_0_1s
@++(590) E0_16100  ; 进出料转移进料爪A电芯冷却时间
LD TR0
AND=(300) H40 &0  ; 3ST_A进料夹爪有料记忆
@MOV(021) &0 E0_16100  ; 进出料转移进料爪A电芯冷却时间
LD TR0
AND>(320) H50 &0  ; 3ST_B进料夹爪有料记忆
AND P_0_1s
@++(590) E0_17100  ; 进出料转移B进料爪电芯冷却时间
LD TR0
AND=(300) H50 &0  ; 3ST_B进料夹爪有料记忆
@MOV(021) &0 E0_17100  ; 进出料转移B进料爪电芯冷却时间

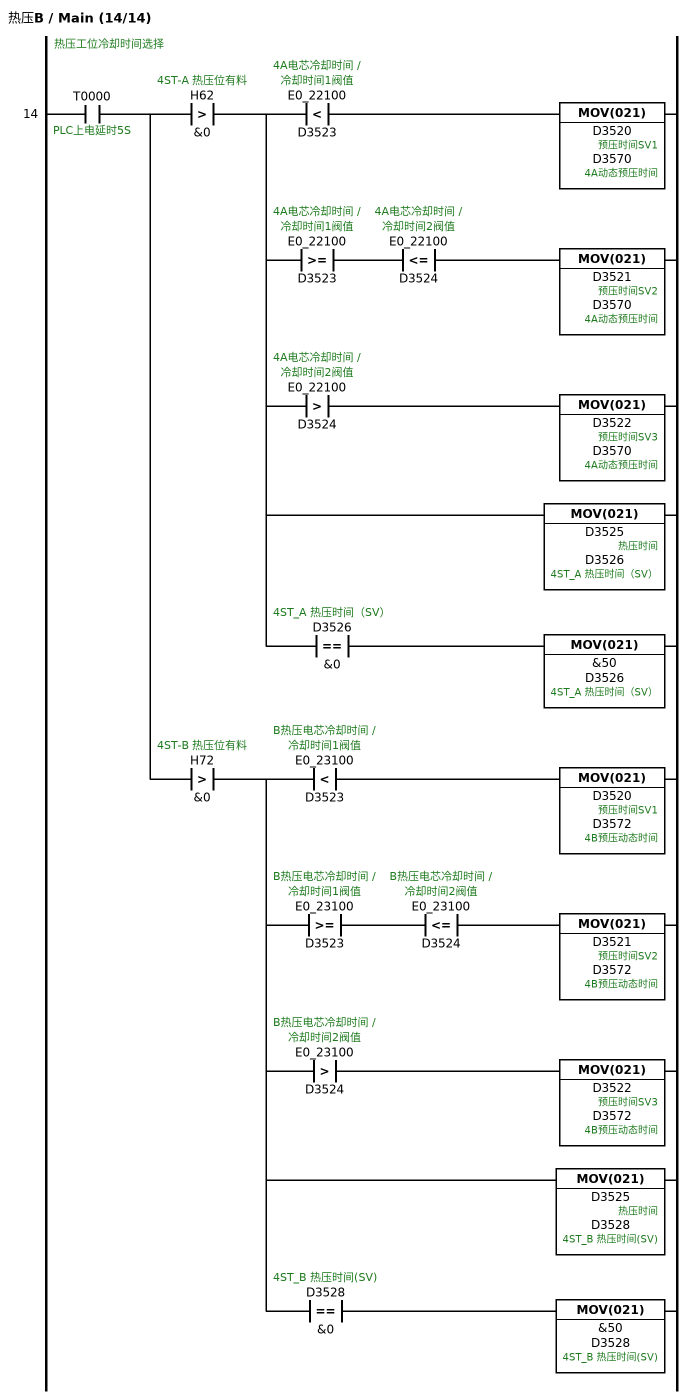
; rung 14: 热压工位冷却时间选择
LD T0000  ; PLC上电延时5S
OUT TR0
AND>(320) H62 &0  ; 4ST-A 热压位有料
OUT TR1
AND<(310) E0_22100 D3523  ; 4A电芯冷却时间, 冷却时间1阀值
MOV(021) D3520 D3570  ; 预压时间SV1, 4A动态预压时间
LD TR1
AND>=(325) E0_22100 D3523  ; 4A电芯冷却时间, 冷却时间1阀值
AND<=(315) E0_22100 D3524  ; 4A电芯冷却时间, 冷却时间2阀值
MOV(021) D3521 D3570  ; 预压时间SV2, 4A动态预压时间
LD TR1
AND>(320) E0_22100 D3524  ; 4A电芯冷却时间, 冷却时间2阀值
MOV(021) D3522 D3570  ; 预压时间SV3, 4A动态预压时间
LD TR1
MOV(021) D3525 D3526  ; 热压时间, 4ST_A 热压时间（SV）
AND=(300) D3526 &0  ; 4ST_A 热压时间（SV）
MOV(021) &50 D3526  ; 4ST_A 热压时间（SV）
LD TR0
AND>(320) H72 &0  ; 4ST-B 热压位有料
OUT TR0
AND<(310) E0_23100 D3523  ; B热压电芯冷却时间, 冷却时间1阀值
MOV(021) D3520 D3572  ; 预压时间SV1, 4B预压动态时间
LD TR0
AND>=(325) E0_23100 D3523  ; B热压电芯冷却时间, 冷却时间1阀值
AND<=(315) E0_23100 D3524  ; B热压电芯冷却时间, 冷却时间2阀值
MOV(021) D3521 D3572  ; 预压时间SV2, 4B预压动态时间
LD TR0
AND>(320) E0_23100 D3524  ; B热压电芯冷却时间, 冷却时间2阀值
MOV(021) D3522 D3572  ; 预压时间SV3, 4B预压动态时间
LD TR0
MOV(021) D3525 D3528  ; 热压时间, 4ST_B 热压时间(SV)
AND=(300) D3528 &0  ; 4ST_B 热压时间(SV)
MOV(021) &50 D3528  ; 4ST_B 热压时间(SV)

### Section _4ST_2热压B

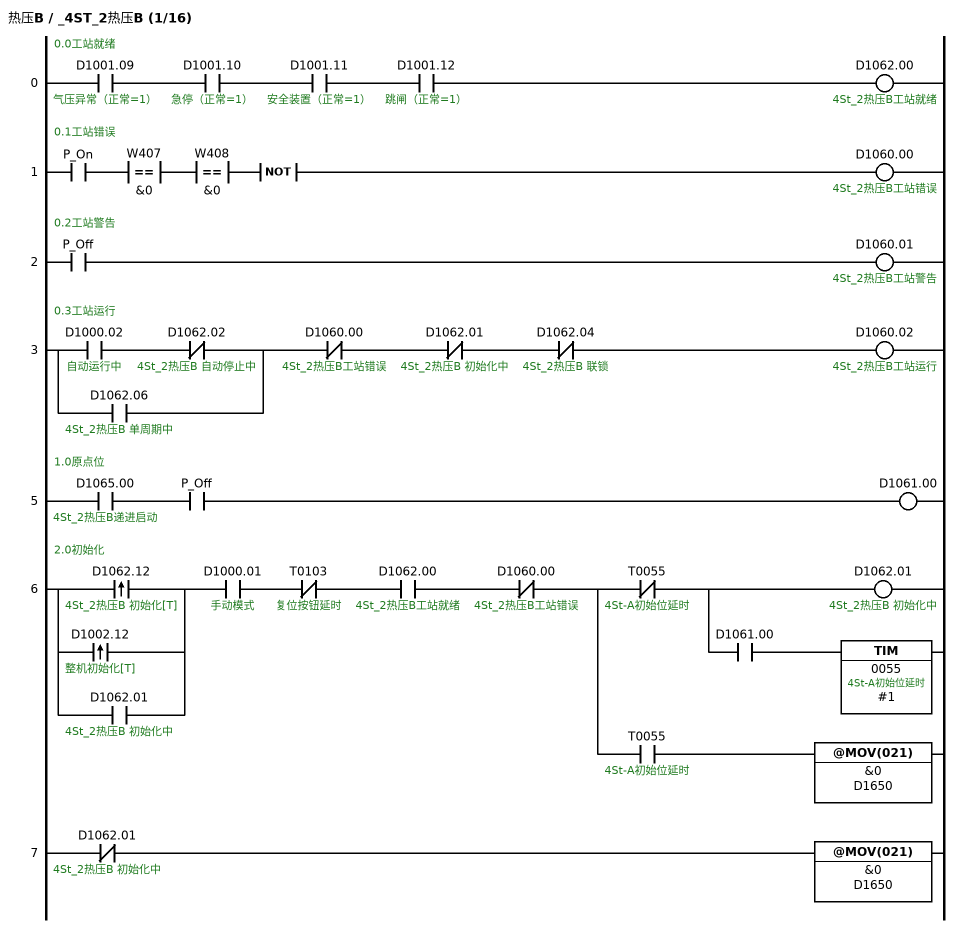
; rung 0: 0.0工站就绪
LD D1001.09  ; 气压异常（正常=1）
AND D1001.10  ; 急停（正常=1）
AND D1001.11  ; 安全装置（正常=1）
AND D1001.12  ; 跳闸（正常=1）
OUT D1062.00  ; 4St_2热压B工站就绪
; rung 1: 0.1工站错误
LD P_On
AND=(300) W407 &0
AND=(300) W408 &0
NOT(520)
OUT D1060.00  ; 4St_2热压B工站错误
; rung 2: 0.2工站警告
LD P_Off
OUT D1060.01  ; 4St_2热压B工站警告
; rung 3: 0.3工站运行
LD D1000.02  ; 自动运行中
ANDNOT D1062.02  ; 4St_2热压B 自动停止中
OR D1062.06  ; 4St_2热压B 单周期中
ANDNOT D1060.00  ; 4St_2热压B工站错误
ANDNOT D1062.01  ; 4St_2热压B 初始化中
ANDNOT D1062.04  ; 4St_2热压B 联锁
OUT D1060.02  ; 4St_2热压B工站运行
; rung 4: 辅助位置
; rung 5: 1.0原点位
LD D1065.00  ; 4St_2热压B递进启动
AND P_Off
OUT D1061.00
; rung 6: 2.0初始化
@LD D1062.12  ; 4St_2热压B 初始化[T]
@OR D1002.12  ; 整机初始化[T]
OR D1062.01  ; 4St_2热压B 初始化中
AND D1000.01  ; 手动模式
ANDNOT T0103  ; 复位按钮延时
AND D1062.00  ; 4St_2热压B工站就绪
ANDNOT D1060.00  ; 4St_2热压B工站错误
OUT TR0
ANDNOT T0055  ; 4St-A初始位延时
OUT D1062.01  ; 4St_2热压B 初始化中
AND D1061.00
TIM 0055 #1  ; 4St-A初始位延时
LD TR0
AND T0055  ; 4St-A初始位延时
@MOV(021) &0 D1650
; rung 7
LDNOT D1062.01  ; 4St_2热压B 初始化中
@MOV(021) &0 D1650

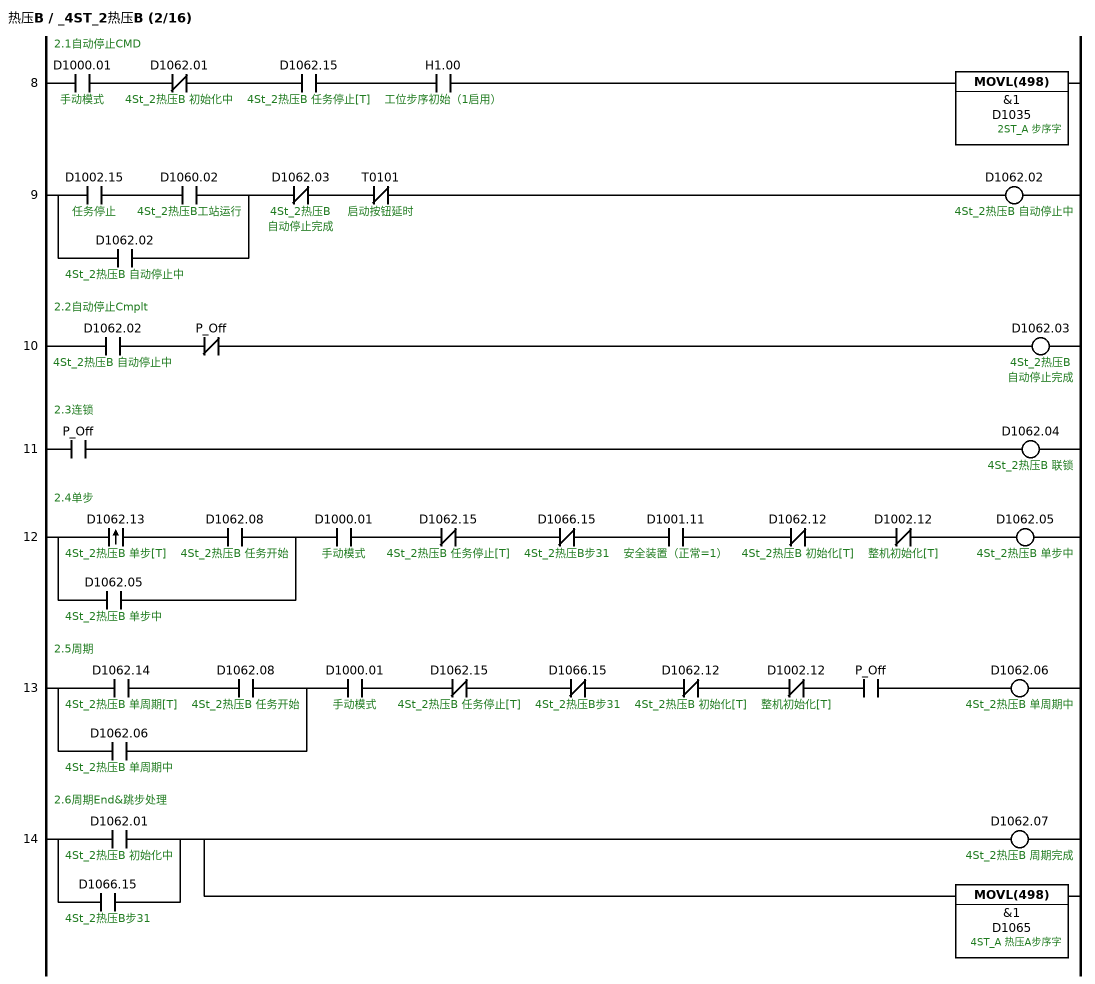
; rung 8: 2.1自动停止CMD
LD D1000.01  ; 手动模式
ANDNOT D1062.01  ; 4St_2热压B 初始化中
AND D1062.15  ; 4St_2热压B 任务停止[T]
AND H1.00  ; 工位步序初始（1启用）
MOVL(498) &1 D1035  ; 2ST_A 步序字
; rung 9
LD D1002.15  ; 任务停止
AND D1060.02  ; 4St_2热压B工站运行
OR D1062.02  ; 4St_2热压B 自动停止中
ANDNOT D1062.03  ; 4St_2热压B 自动停止完成
ANDNOT T0101  ; 启动按钮延时
OUT D1062.02  ; 4St_2热压B 自动停止中
; rung 10: 2.2自动停止Cmplt
LD D1062.02  ; 4St_2热压B 自动停止中
ANDNOT P_Off
OUT D1062.03  ; 4St_2热压B 自动停止完成
; rung 11: 2.3连锁
LD P_Off
OUT D1062.04  ; 4St_2热压B 联锁
; rung 12: 2.4单步
@LD D1062.13  ; 4St_2热压B 单步[T]
AND D1062.08  ; 4St_2热压B 任务开始
OR D1062.05  ; 4St_2热压B 单步中
AND D1000.01  ; 手动模式
ANDNOT D1062.15  ; 4St_2热压B 任务停止[T]
ANDNOT D1066.15  ; 4St_2热压B步31
AND D1001.11  ; 安全装置（正常=1）
ANDNOT D1062.12  ; 4St_2热压B 初始化[T]
ANDNOT D1002.12  ; 整机初始化[T]
OUT D1062.05  ; 4St_2热压B 单步中
; rung 13: 2.5周期
LD D1062.14  ; 4St_2热压B 单周期[T]
AND D1062.08  ; 4St_2热压B 任务开始
OR D1062.06  ; 4St_2热压B 单周期中
AND D1000.01  ; 手动模式
ANDNOT D1062.15  ; 4St_2热压B 任务停止[T]
ANDNOT D1066.15  ; 4St_2热压B步31
ANDNOT D1062.12  ; 4St_2热压B 初始化[T]
ANDNOT D1002.12  ; 整机初始化[T]
AND P_Off
OUT D1062.06  ; 4St_2热压B 单周期中
; rung 14: 2.6周期End&跳步处理
LD D1062.01  ; 4St_2热压B 初始化中
OR D1066.15  ; 4St_2热压B步31
OUT D1062.07  ; 4St_2热压B 周期完成
MOVL(498) &1 D1065  ; 4ST_A 热压A步序字

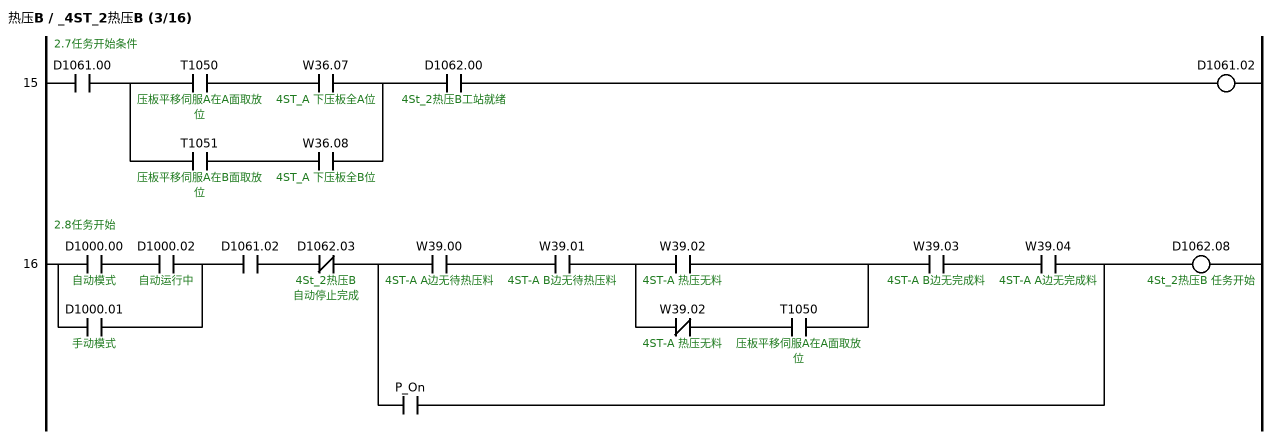
; rung 15: 2.7任务开始条件
LD D1061.00
LD T1050  ; 压板平移伺服A在A面取放位
AND W36.07  ; 4ST_A 下压板全A位
LD T1051  ; 压板平移伺服A在B面取放位
AND W36.08  ; 4ST_A 下压板全B位
ORLD
ANDLD
AND D1062.00  ; 4St_2热压B工站就绪
OUT D1061.02
; rung 16: 2.8任务开始
LD D1000.00  ; 自动模式
AND D1000.02  ; 自动运行中
OR D1000.01  ; 手动模式
AND D1061.02
ANDNOT D1062.03  ; 4St_2热压B 自动停止完成
LD W39.00  ; 4ST-A A边无待热压料
AND W39.01  ; 4ST-A B边无待热压料
LD W39.02  ; 4ST-A 热压无料
LDNOT W39.02  ; 4ST-A 热压无料
AND T1050  ; 压板平移伺服A在A面取放位
ORLD
ANDLD
AND W39.03  ; 4ST-A B边无完成料
AND W39.04  ; 4ST-A A边无完成料
OR P_On
ANDLD
OUT D1062.08  ; 4St_2热压B 任务开始

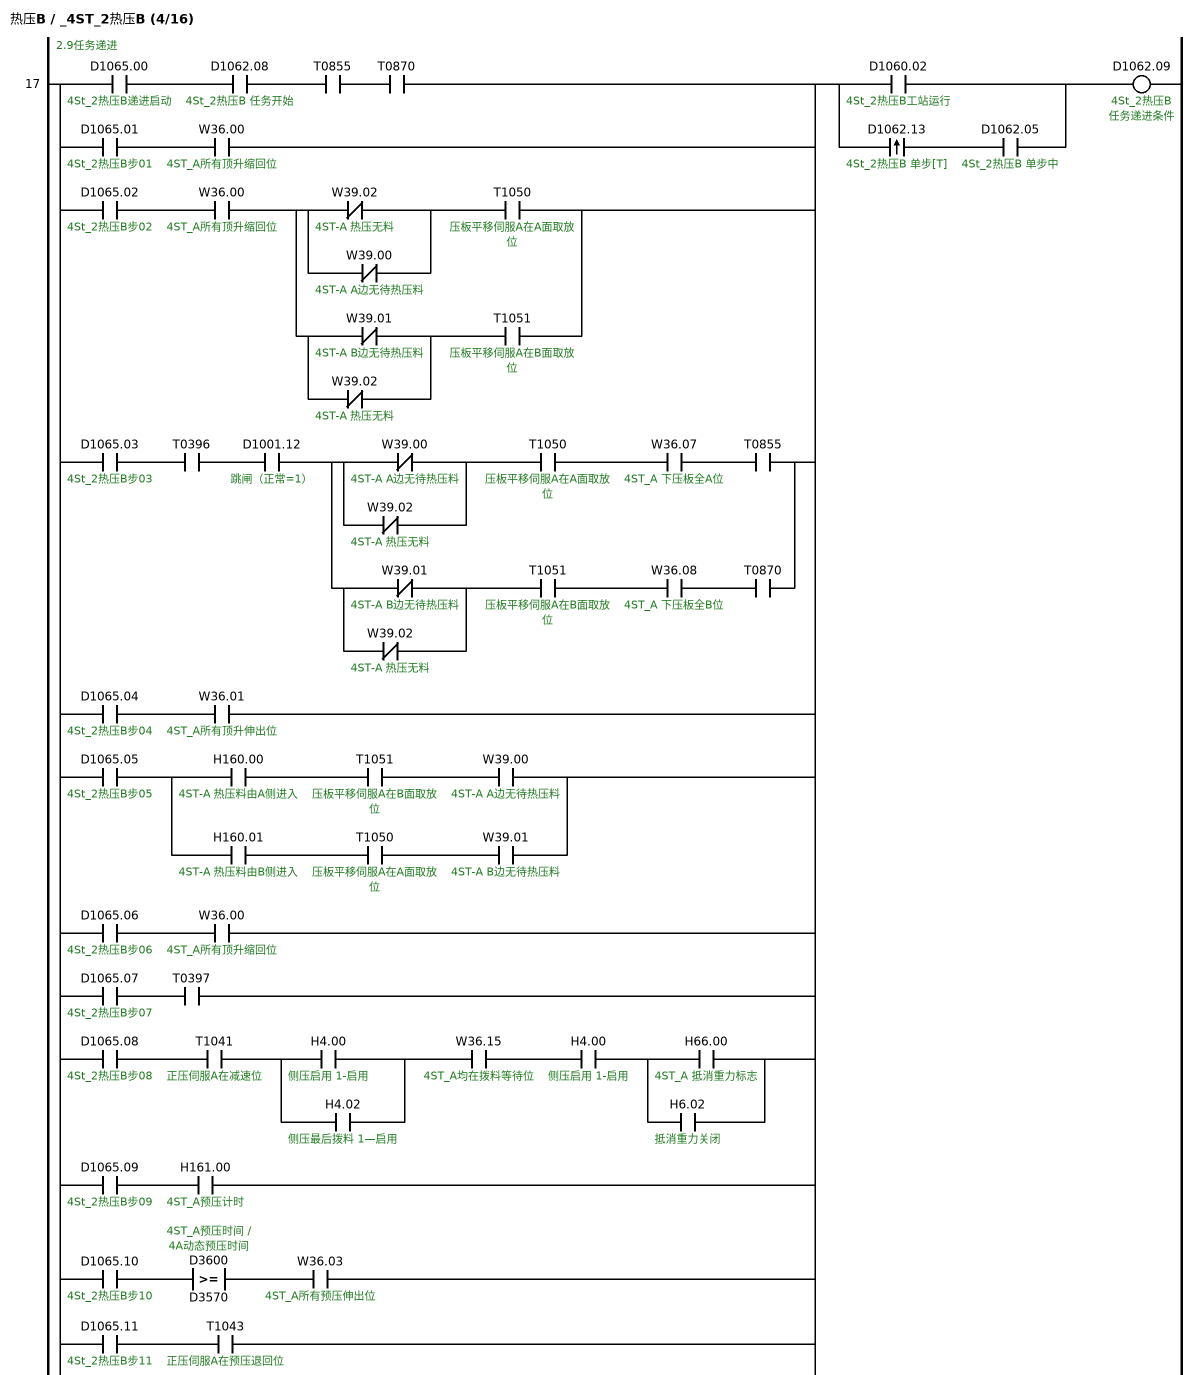

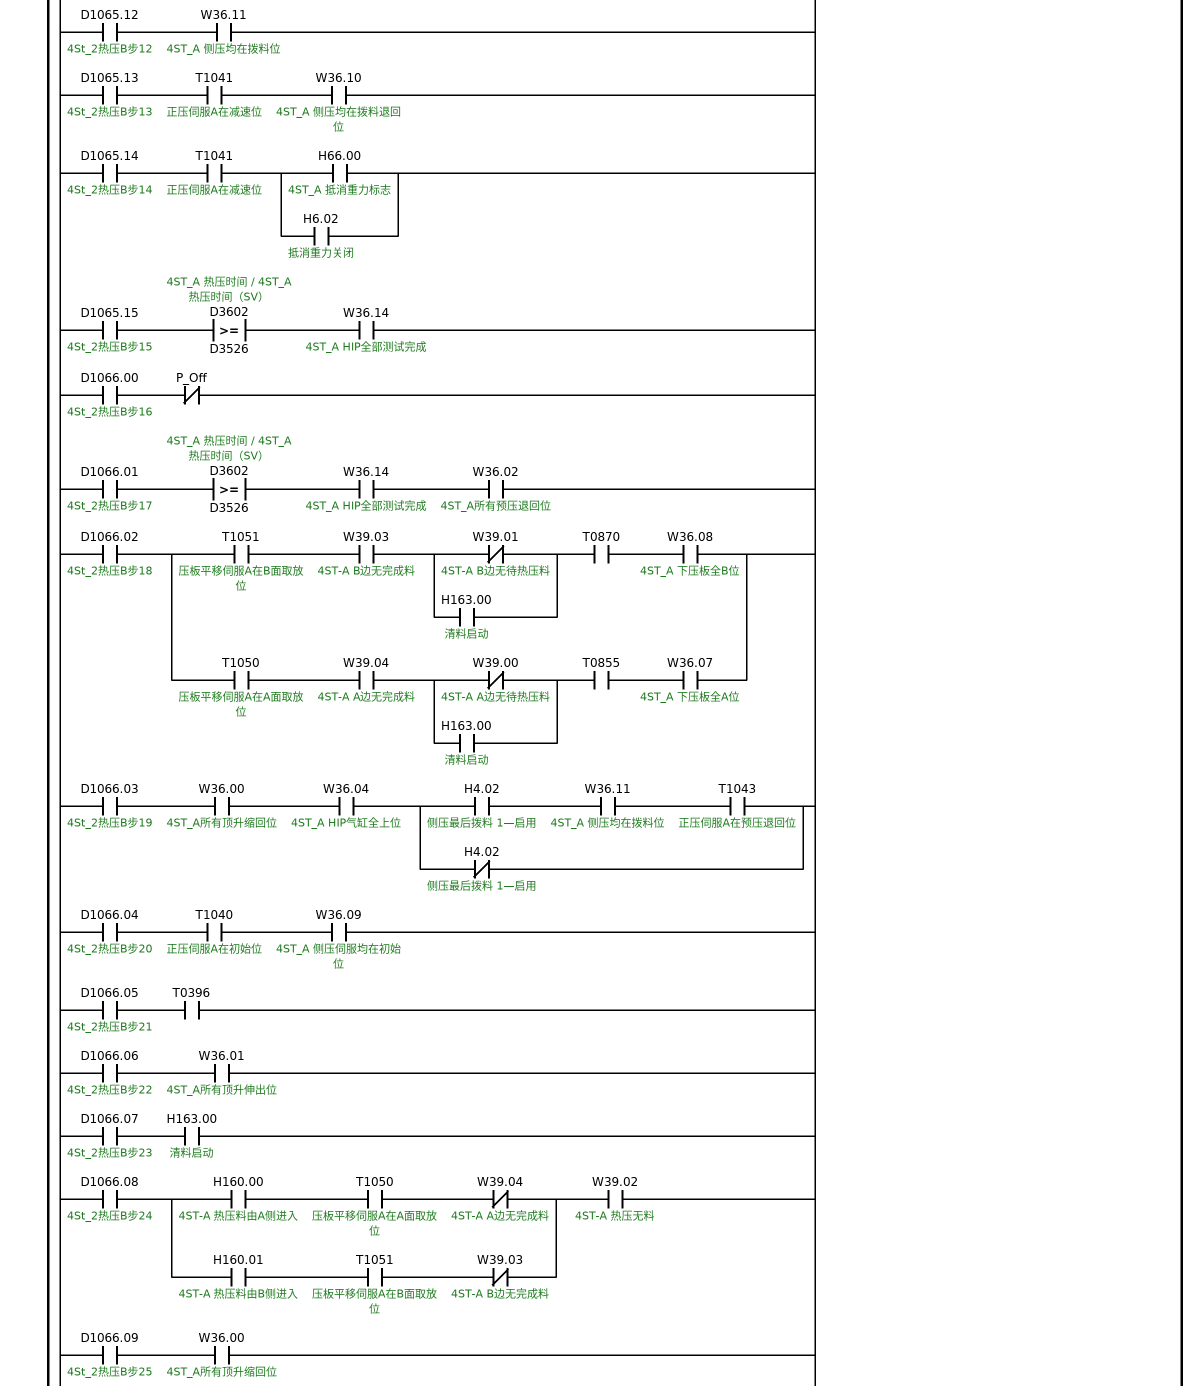

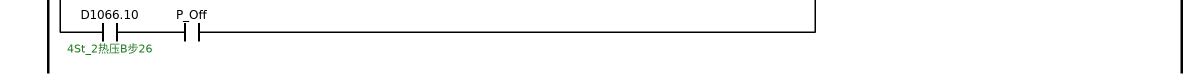
; rung 17: 2.9任务递进
LD D1065.00  ; 4St_2热压B递进启动
AND D1062.08  ; 4St_2热压B 任务开始
AND T0855
AND T0870
LD D1065.01  ; 4St_2热压B步01
AND W36.00  ; 4ST_A所有顶升缩回位
ORLD
LD D1065.02  ; 4St_2热压B步02
AND W36.00  ; 4ST_A所有顶升缩回位
LDNOT W39.02  ; 4ST-A 热压无料
ORNOT W39.00  ; 4ST-A A边无待热压料
AND T1050  ; 压板平移伺服A在A面取放位
LDNOT W39.01  ; 4ST-A B边无待热压料
ORNOT W39.02  ; 4ST-A 热压无料
AND T1051  ; 压板平移伺服A在B面取放位
ORLD
ANDLD
ORLD
LD D1065.03  ; 4St_2热压B步03
AND T0396
AND D1001.12  ; 跳闸（正常=1）
LDNOT W39.00  ; 4ST-A A边无待热压料
ORNOT W39.02  ; 4ST-A 热压无料
AND T1050  ; 压板平移伺服A在A面取放位
AND W36.07  ; 4ST_A 下压板全A位
AND T0855
LDNOT W39.01  ; 4ST-A B边无待热压料
ORNOT W39.02  ; 4ST-A 热压无料
AND T1051  ; 压板平移伺服A在B面取放位
AND W36.08  ; 4ST_A 下压板全B位
AND T0870
ORLD
ANDLD
ORLD
LD D1065.04  ; 4St_2热压B步04
AND W36.01  ; 4ST_A所有顶升伸出位
ORLD
LD D1065.05  ; 4St_2热压B步05
LD H160.00  ; 4ST-A 热压料由A侧进入
AND T1051  ; 压板平移伺服A在B面取放位
AND W39.00  ; 4ST-A A边无待热压料
LD H160.01  ; 4ST-A 热压料由B侧进入
AND T1050  ; 压板平移伺服A在A面取放位
AND W39.01  ; 4ST-A B边无待热压料
ORLD
ANDLD
ORLD
LD D1065.06  ; 4St_2热压B步06
AND W36.00  ; 4ST_A所有顶升缩回位
ORLD
LD D1065.07  ; 4St_2热压B步07
AND T0397
ORLD
LD D1065.08  ; 4St_2热压B步08
AND T1041  ; 正压伺服A在减速位
LD H4.00  ; 侧压启用 1-启用
OR H4.02  ; 侧压最后拨料 1—启用
ANDLD
AND W36.15  ; 4ST_A均在拨料等待位
AND H4.00  ; 侧压启用 1-启用
LD H66.00  ; 4ST_A 抵消重力标志
OR H6.02  ; 抵消重力关闭
ANDLD
ORLD
LD D1065.09  ; 4St_2热压B步09
AND H161.00  ; 4ST_A预压计时
ORLD
LD D1065.10  ; 4St_2热压B步10
AND>=(325) D3600 D3570  ; 4ST_A预压时间, 4A动态预压时间
AND W36.03  ; 4ST_A所有预压伸出位
ORLD
LD D1065.11  ; 4St_2热压B步11
AND T1043  ; 正压伺服A在预压退回位
ORLD
LD D1065.12  ; 4St_2热压B步12
AND W36.11  ; 4ST_A 侧压均在拨料位
ORLD
LD D1065.13  ; 4St_2热压B步13
AND T1041  ; 正压伺服A在减速位
AND W36.10  ; 4ST_A 侧压均在拨料退回位
ORLD
LD D1065.14  ; 4St_2热压B步14
AND T1041  ; 正压伺服A在减速位
LD H66.00  ; 4ST_A 抵消重力标志
OR H6.02  ; 抵消重力关闭
ANDLD
ORLD
LD D1065.15  ; 4St_2热压B步15
AND>=(325) D3602 D3526  ; 4ST_A 热压时间, 4ST_A 热压时间（SV）
AND W36.14  ; 4ST_A HIP全部测试完成
ORLD
LD D1066.00  ; 4St_2热压B步16
ANDNOT P_Off
ORLD
LD D1066.01  ; 4St_2热压B步17
AND>=(325) D3602 D3526  ; 4ST_A 热压时间, 4ST_A 热压时间（SV）
AND W36.14  ; 4ST_A HIP全部测试完成
AND W36.02  ; 4ST_A所有预压退回位
ORLD
LD D1066.02  ; 4St_2热压B步18
LD T1051  ; 压板平移伺服A在B面取放位
AND W39.03  ; 4ST-A B边无完成料
LDNOT W39.01  ; 4ST-A B边无待热压料
OR H163.00  ; 清料启动
ANDLD
AND T0870
AND W36.08  ; 4ST_A 下压板全B位
LD T1050  ; 压板平移伺服A在A面取放位
AND W39.04  ; 4ST-A A边无完成料
LDNOT W39.00  ; 4ST-A A边无待热压料
OR H163.00  ; 清料启动
ANDLD
AND T0855
AND W36.07  ; 4ST_A 下压板全A位
ORLD
ANDLD
ORLD
LD D1066.03  ; 4St_2热压B步19
AND W36.00  ; 4ST_A所有顶升缩回位
AND W36.04  ; 4ST_A HIP气缸全上位
LD H4.02  ; 侧压最后拨料 1—启用
AND W36.11  ; 4ST_A 侧压均在拨料位
AND T1043  ; 正压伺服A在预压退回位
ORNOT H4.02  ; 侧压最后拨料 1—启用
ANDLD
ORLD
LD D1066.04  ; 4St_2热压B步20
AND T1040  ; 正压伺服A在初始位
AND W36.09  ; 4ST_A 侧压伺服均在初始位
ORLD
LD D1066.05  ; 4St_2热压B步21
AND T0396
ORLD
LD D1066.06  ; 4St_2热压B步22
AND W36.01  ; 4ST_A所有顶升伸出位
ORLD
LD D1066.07  ; 4St_2热压B步23
AND H163.00  ; 清料启动
ORLD
LD D1066.08  ; 4St_2热压B步24
LD H160.00  ; 4ST-A 热压料由A侧进入
AND T1050  ; 压板平移伺服A在A面取放位
ANDNOT W39.04  ; 4ST-A A边无完成料
LD H160.01  ; 4ST-A 热压料由B侧进入
AND T1051  ; 压板平移伺服A在B面取放位
ANDNOT W39.03  ; 4ST-A B边无完成料
ORLD
ANDLD
AND W39.02  ; 4ST-A 热压无料
ORLD
LD D1066.09  ; 4St_2热压B步25
AND W36.00  ; 4ST_A所有顶升缩回位
ORLD
LD D1066.10  ; 4St_2热压B步26
AND P_Off
ORLD
LD D1060.02  ; 4St_2热压B工站运行
@LD D1062.13  ; 4St_2热压B 单步[T]
AND D1062.05  ; 4St_2热压B 单步中
ORLD
ANDLD
OUT D1062.09  ; 4St_2热压B 任务递进条件

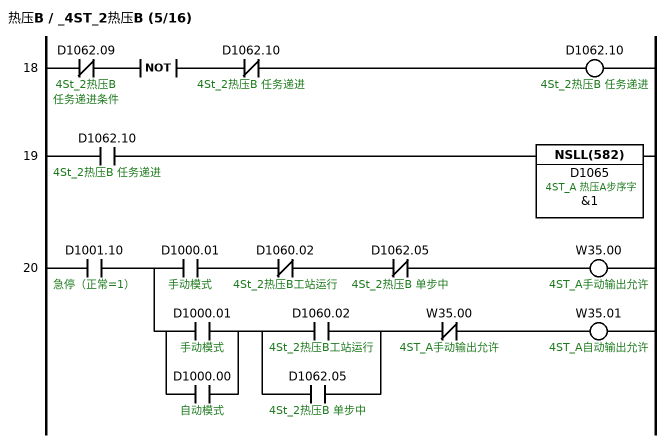
; rung 18
LDNOT D1062.09  ; 4St_2热压B 任务递进条件
NOT(520)
ANDNOT D1062.10  ; 4St_2热压B 任务递进
OUT D1062.10  ; 4St_2热压B 任务递进
; rung 19
LD D1062.10  ; 4St_2热压B 任务递进
NSLL(582) D1065 &1  ; 4ST_A 热压A步序字
; rung 20
LD D1001.10  ; 急停（正常=1）
OUT TR0
AND D1000.01  ; 手动模式
ANDNOT D1060.02  ; 4St_2热压B工站运行
ANDNOT D1062.05  ; 4St_2热压B 单步中
OUT W35.00  ; 4ST_A手动输出允许
LD TR0
LD D1000.01  ; 手动模式
OR D1000.00  ; 自动模式
ANDLD
LD D1060.02  ; 4St_2热压B工站运行
OR D1062.05  ; 4St_2热压B 单步中
ANDLD
ANDNOT W35.00  ; 4ST_A手动输出允许
OUT W35.01  ; 4ST_A自动输出允许

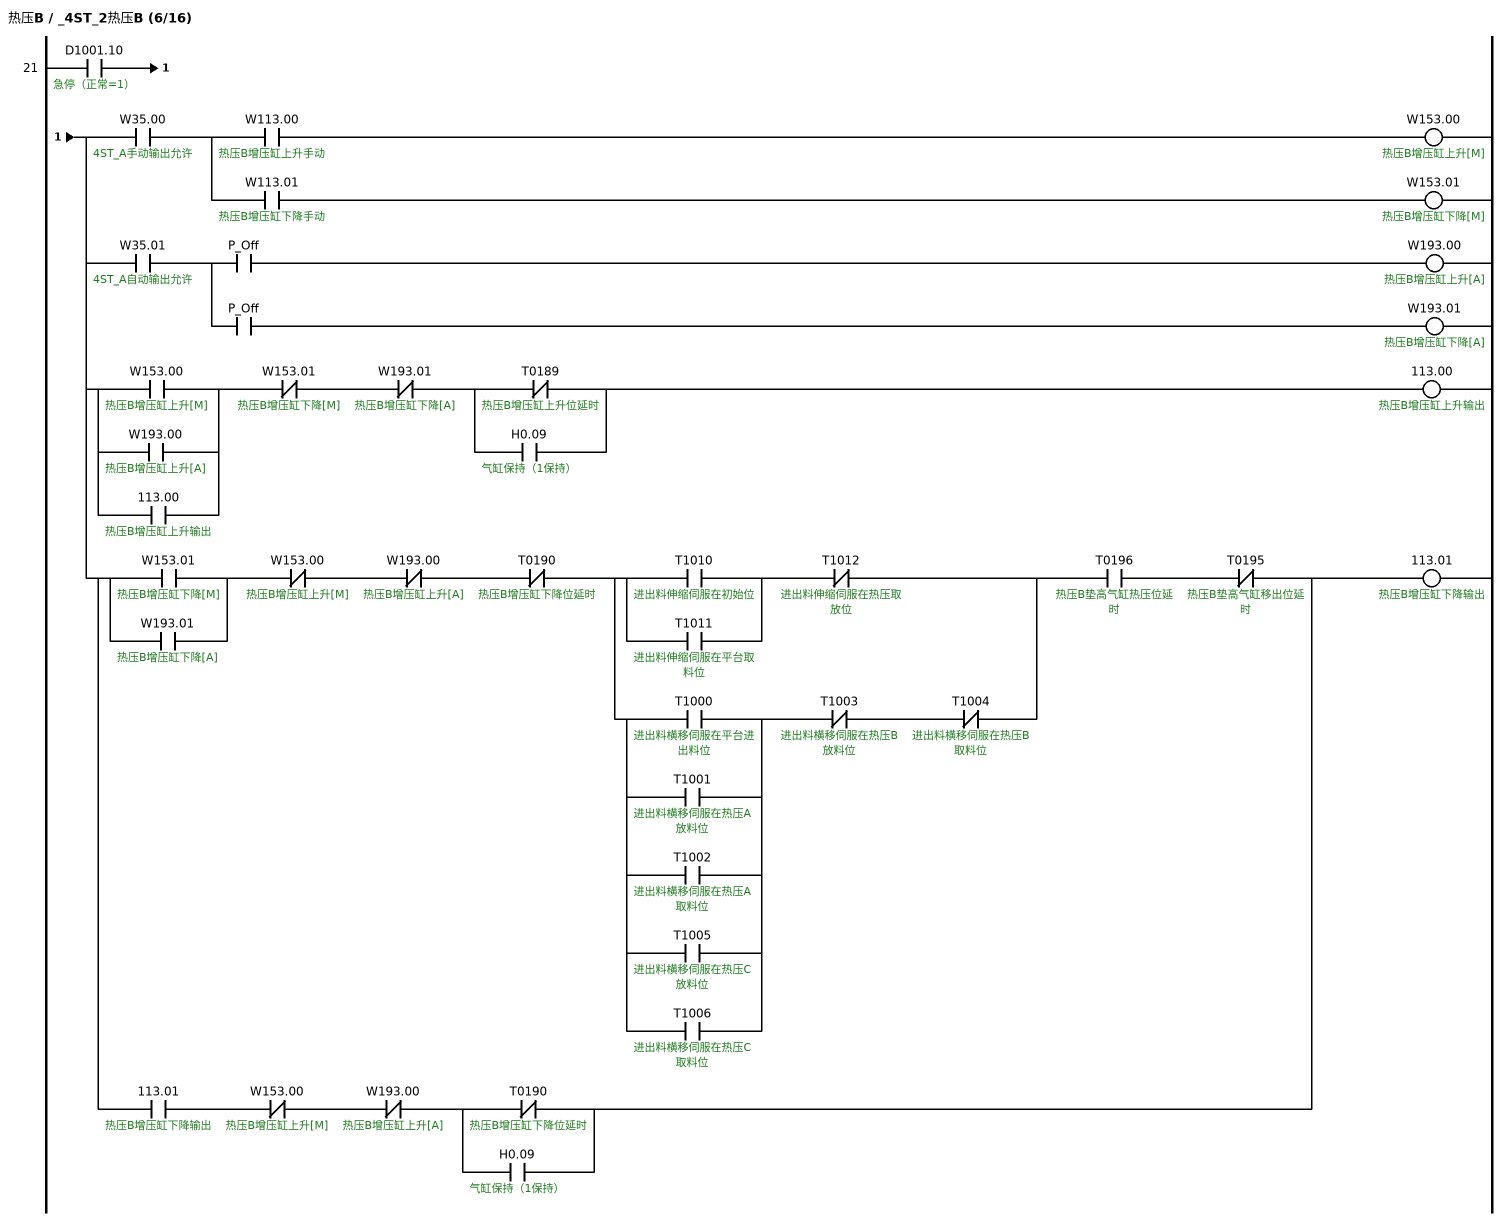
; rung 21
LD D1001.10  ; 急停（正常=1）
OUT TR0
AND W35.00  ; 4ST_A手动输出允许
OUT TR1
AND W113.00  ; 热压B增压缸上升手动
OUT W153.00  ; 热压B增压缸上升[M]
LD TR1
AND W113.01  ; 热压B增压缸下降手动
OUT W153.01  ; 热压B增压缸下降[M]
LD TR0
AND W35.01  ; 4ST_A自动输出允许
OUT TR1
AND P_Off
OUT W193.00  ; 热压B增压缸上升[A]
LD TR1
AND P_Off
OUT W193.01  ; 热压B增压缸下降[A]
LD TR0
LD W153.00  ; 热压B增压缸上升[M]
OR W193.00  ; 热压B增压缸上升[A]
OR 113.00  ; 热压B增压缸上升输出
ANDLD
ANDNOT W153.01  ; 热压B增压缸下降[M]
ANDNOT W193.01  ; 热压B增压缸下降[A]
LDNOT T0189  ; 热压B增压缸上升位延时
OR H0.09  ; 气缸保持（1保持）
ANDLD
OUT 113.00  ; 热压B增压缸上升输出
LD TR0
LD W153.01  ; 热压B增压缸下降[M]
OR W193.01  ; 热压B增压缸下降[A]
ANDNOT W153.00  ; 热压B增压缸上升[M]
ANDNOT W193.00  ; 热压B增压缸上升[A]
ANDNOT T0190  ; 热压B增压缸下降位延时
LD T1010  ; 进出料伸缩伺服在初始位
OR T1011  ; 进出料伸缩伺服在平台取料位
ANDNOT T1012  ; 进出料伸缩伺服在热压取放位
LD T1000  ; 进出料横移伺服在平台进出料位
OR T1001  ; 进出料横移伺服在热压A放料位
OR T1002  ; 进出料横移伺服在热压A取料位
OR T1005  ; 进出料横移伺服在热压C放料位
OR T1006  ; 进出料横移伺服在热压C取料位
ANDNOT T1003  ; 进出料横移伺服在热压B放料位
ANDNOT T1004  ; 进出料横移伺服在热压B取料位
ORLD
ANDLD
AND T0196  ; 热压B垫高气缸热压位延时
ANDNOT T0195  ; 热压B垫高气缸移出位延时
LD 113.01  ; 热压B增压缸下降输出
ANDNOT W153.00  ; 热压B增压缸上升[M]
ANDNOT W193.00  ; 热压B增压缸上升[A]
LDNOT T0190  ; 热压B增压缸下降位延时
OR H0.09  ; 气缸保持（1保持）
ANDLD
ORLD
ANDLD
OUT 113.01  ; 热压B增压缸下降输出

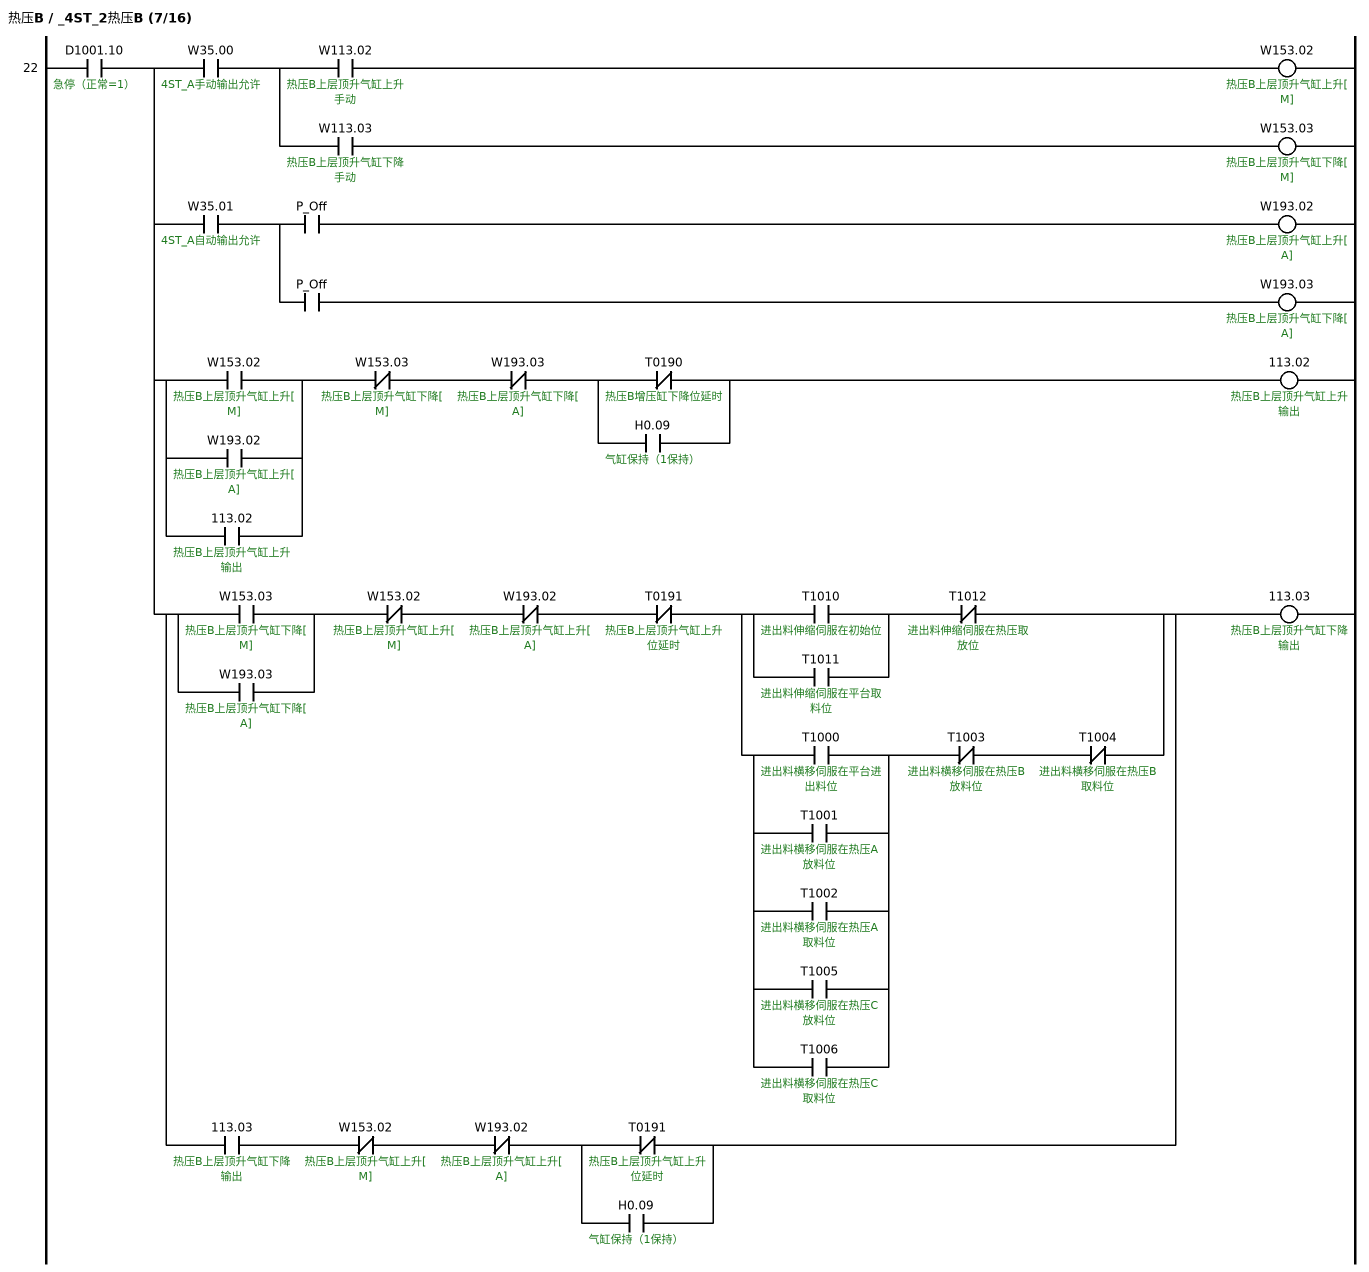
; rung 22
LD D1001.10  ; 急停（正常=1）
OUT TR0
AND W35.00  ; 4ST_A手动输出允许
OUT TR1
AND W113.02  ; 热压B上层顶升气缸上升手动
OUT W153.02  ; 热压B上层顶升气缸上升[M]
LD TR1
AND W113.03  ; 热压B上层顶升气缸下降手动
OUT W153.03  ; 热压B上层顶升气缸下降[M]
LD TR0
AND W35.01  ; 4ST_A自动输出允许
OUT TR1
AND P_Off
OUT W193.02  ; 热压B上层顶升气缸上升[A]
LD TR1
AND P_Off
OUT W193.03  ; 热压B上层顶升气缸下降[A]
LD TR0
LD W153.02  ; 热压B上层顶升气缸上升[M]
OR W193.02  ; 热压B上层顶升气缸上升[A]
OR 113.02  ; 热压B上层顶升气缸上升输出
ANDLD
ANDNOT W153.03  ; 热压B上层顶升气缸下降[M]
ANDNOT W193.03  ; 热压B上层顶升气缸下降[A]
LDNOT T0190  ; 热压B增压缸下降位延时
OR H0.09  ; 气缸保持（1保持）
ANDLD
OUT 113.02  ; 热压B上层顶升气缸上升输出
LD TR0
LD W153.03  ; 热压B上层顶升气缸下降[M]
OR W193.03  ; 热压B上层顶升气缸下降[A]
ANDNOT W153.02  ; 热压B上层顶升气缸上升[M]
ANDNOT W193.02  ; 热压B上层顶升气缸上升[A]
ANDNOT T0191  ; 热压B上层顶升气缸上升位延时
LD T1010  ; 进出料伸缩伺服在初始位
OR T1011  ; 进出料伸缩伺服在平台取料位
ANDNOT T1012  ; 进出料伸缩伺服在热压取放位
LD T1000  ; 进出料横移伺服在平台进出料位
OR T1001  ; 进出料横移伺服在热压A放料位
OR T1002  ; 进出料横移伺服在热压A取料位
OR T1005  ; 进出料横移伺服在热压C放料位
OR T1006  ; 进出料横移伺服在热压C取料位
ANDNOT T1003  ; 进出料横移伺服在热压B放料位
ANDNOT T1004  ; 进出料横移伺服在热压B取料位
ORLD
ANDLD
LD 113.03  ; 热压B上层顶升气缸下降输出
ANDNOT W153.02  ; 热压B上层顶升气缸上升[M]
ANDNOT W193.02  ; 热压B上层顶升气缸上升[A]
LDNOT T0191  ; 热压B上层顶升气缸上升位延时
OR H0.09  ; 气缸保持（1保持）
ANDLD
ORLD
ANDLD
OUT 113.03  ; 热压B上层顶升气缸下降输出

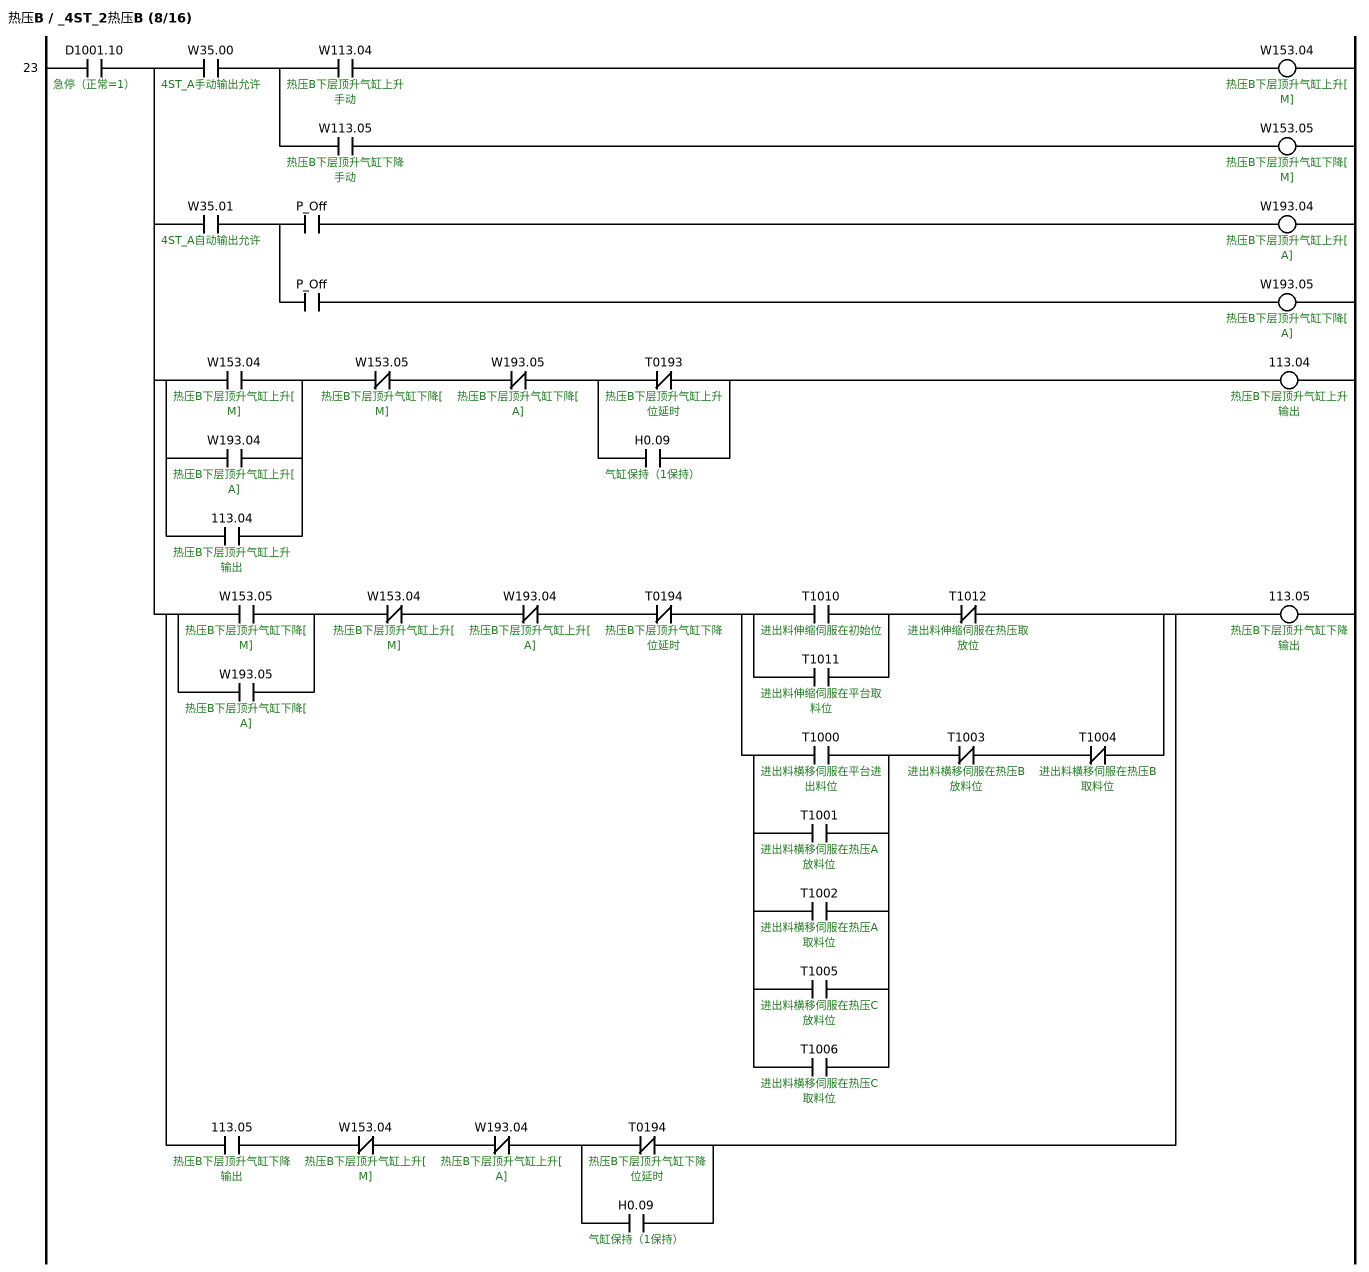
; rung 23
LD D1001.10  ; 急停（正常=1）
OUT TR0
AND W35.00  ; 4ST_A手动输出允许
OUT TR1
AND W113.04  ; 热压B下层顶升气缸上升手动
OUT W153.04  ; 热压B下层顶升气缸上升[M]
LD TR1
AND W113.05  ; 热压B下层顶升气缸下降手动
OUT W153.05  ; 热压B下层顶升气缸下降[M]
LD TR0
AND W35.01  ; 4ST_A自动输出允许
OUT TR1
AND P_Off
OUT W193.04  ; 热压B下层顶升气缸上升[A]
LD TR1
AND P_Off
OUT W193.05  ; 热压B下层顶升气缸下降[A]
LD TR0
LD W153.04  ; 热压B下层顶升气缸上升[M]
OR W193.04  ; 热压B下层顶升气缸上升[A]
OR 113.04  ; 热压B下层顶升气缸上升输出
ANDLD
ANDNOT W153.05  ; 热压B下层顶升气缸下降[M]
ANDNOT W193.05  ; 热压B下层顶升气缸下降[A]
LDNOT T0193  ; 热压B下层顶升气缸上升位延时
OR H0.09  ; 气缸保持（1保持）
ANDLD
OUT 113.04  ; 热压B下层顶升气缸上升输出
LD TR0
LD W153.05  ; 热压B下层顶升气缸下降[M]
OR W193.05  ; 热压B下层顶升气缸下降[A]
ANDNOT W153.04  ; 热压B下层顶升气缸上升[M]
ANDNOT W193.04  ; 热压B下层顶升气缸上升[A]
ANDNOT T0194  ; 热压B下层顶升气缸下降位延时
LD T1010  ; 进出料伸缩伺服在初始位
OR T1011  ; 进出料伸缩伺服在平台取料位
ANDNOT T1012  ; 进出料伸缩伺服在热压取放位
LD T1000  ; 进出料横移伺服在平台进出料位
OR T1001  ; 进出料横移伺服在热压A放料位
OR T1002  ; 进出料横移伺服在热压A取料位
OR T1005  ; 进出料横移伺服在热压C放料位
OR T1006  ; 进出料横移伺服在热压C取料位
ANDNOT T1003  ; 进出料横移伺服在热压B放料位
ANDNOT T1004  ; 进出料横移伺服在热压B取料位
ORLD
ANDLD
LD 113.05  ; 热压B下层顶升气缸下降输出
ANDNOT W153.04  ; 热压B下层顶升气缸上升[M]
ANDNOT W193.04  ; 热压B下层顶升气缸上升[A]
LDNOT T0194  ; 热压B下层顶升气缸下降位延时
OR H0.09  ; 气缸保持（1保持）
ANDLD
ORLD
ANDLD
OUT 113.05  ; 热压B下层顶升气缸下降输出

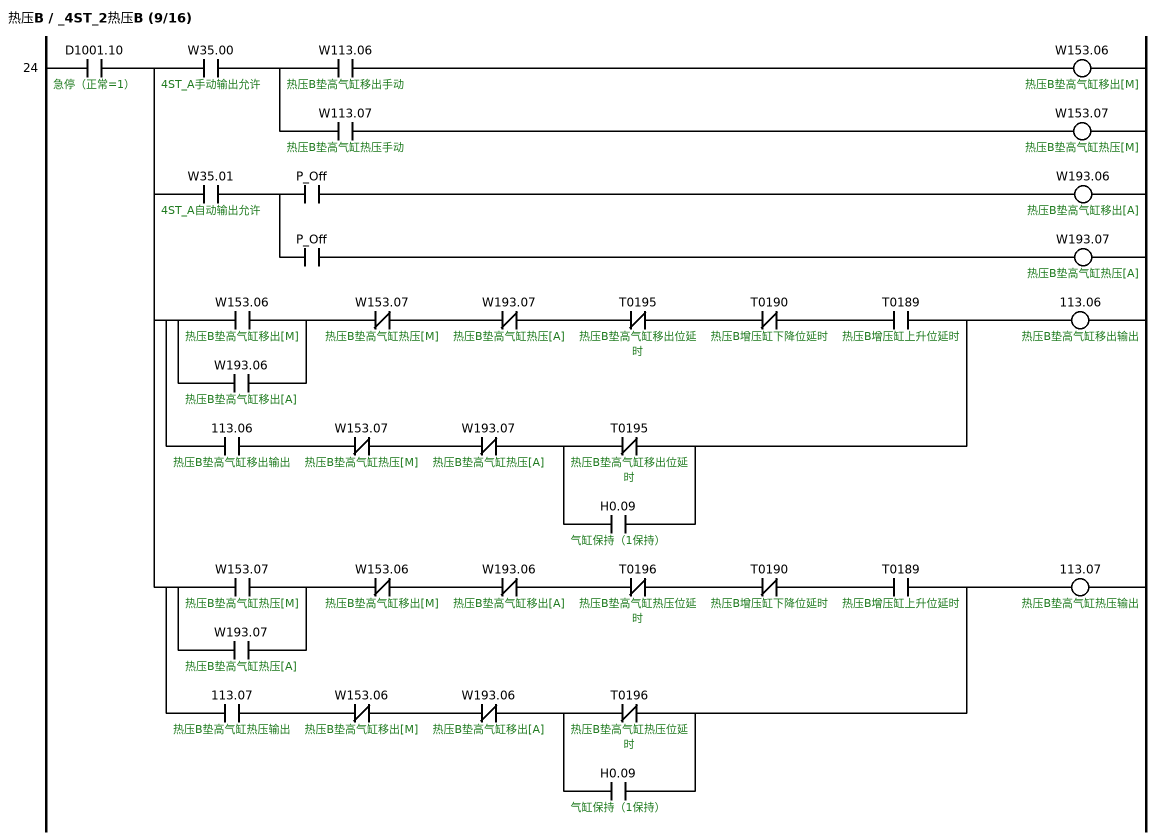
; rung 24
LD D1001.10  ; 急停（正常=1）
OUT TR0
AND W35.00  ; 4ST_A手动输出允许
OUT TR1
AND W113.06  ; 热压B垫高气缸移出手动
OUT W153.06  ; 热压B垫高气缸移出[M]
LD TR1
AND W113.07  ; 热压B垫高气缸热压手动
OUT W153.07  ; 热压B垫高气缸热压[M]
LD TR0
AND W35.01  ; 4ST_A自动输出允许
OUT TR1
AND P_Off
OUT W193.06  ; 热压B垫高气缸移出[A]
LD TR1
AND P_Off
OUT W193.07  ; 热压B垫高气缸热压[A]
LD TR0
LD W153.06  ; 热压B垫高气缸移出[M]
OR W193.06  ; 热压B垫高气缸移出[A]
ANDNOT W153.07  ; 热压B垫高气缸热压[M]
ANDNOT W193.07  ; 热压B垫高气缸热压[A]
ANDNOT T0195  ; 热压B垫高气缸移出位延时
ANDNOT T0190  ; 热压B增压缸下降位延时
AND T0189  ; 热压B增压缸上升位延时
LD 113.06  ; 热压B垫高气缸移出输出
ANDNOT W153.07  ; 热压B垫高气缸热压[M]
ANDNOT W193.07  ; 热压B垫高气缸热压[A]
LDNOT T0195  ; 热压B垫高气缸移出位延时
OR H0.09  ; 气缸保持（1保持）
ANDLD
ORLD
ANDLD
OUT 113.06  ; 热压B垫高气缸移出输出
LD TR0
LD W153.07  ; 热压B垫高气缸热压[M]
OR W193.07  ; 热压B垫高气缸热压[A]
ANDNOT W153.06  ; 热压B垫高气缸移出[M]
ANDNOT W193.06  ; 热压B垫高气缸移出[A]
ANDNOT T0196  ; 热压B垫高气缸热压位延时
ANDNOT T0190  ; 热压B增压缸下降位延时
AND T0189  ; 热压B增压缸上升位延时
LD 113.07  ; 热压B垫高气缸热压输出
ANDNOT W153.06  ; 热压B垫高气缸移出[M]
ANDNOT W193.06  ; 热压B垫高气缸移出[A]
LDNOT T0196  ; 热压B垫高气缸热压位延时
OR H0.09  ; 气缸保持（1保持）
ANDLD
ORLD
ANDLD
OUT 113.07  ; 热压B垫高气缸热压输出

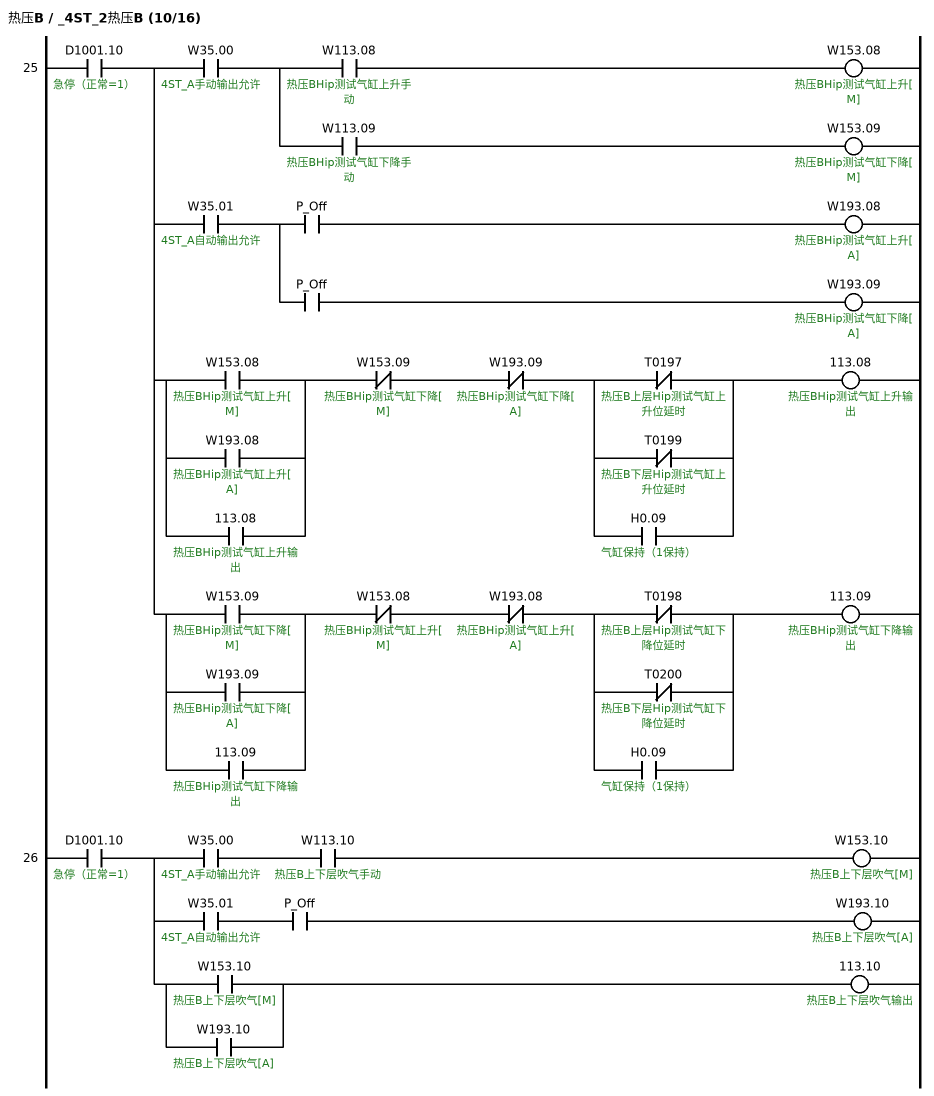
; rung 25
LD D1001.10  ; 急停（正常=1）
OUT TR0
AND W35.00  ; 4ST_A手动输出允许
OUT TR1
AND W113.08  ; 热压BHip测试气缸上升手动
OUT W153.08  ; 热压BHip测试气缸上升[M]
LD TR1
AND W113.09  ; 热压BHip测试气缸下降手动
OUT W153.09  ; 热压BHip测试气缸下降[M]
LD TR0
AND W35.01  ; 4ST_A自动输出允许
OUT TR1
AND P_Off
OUT W193.08  ; 热压BHip测试气缸上升[A]
LD TR1
AND P_Off
OUT W193.09  ; 热压BHip测试气缸下降[A]
LD TR0
LD W153.08  ; 热压BHip测试气缸上升[M]
OR W193.08  ; 热压BHip测试气缸上升[A]
OR 113.08  ; 热压BHip测试气缸上升输出
ANDLD
ANDNOT W153.09  ; 热压BHip测试气缸下降[M]
ANDNOT W193.09  ; 热压BHip测试气缸下降[A]
LDNOT T0197  ; 热压B上层Hip测试气缸上升位延时
ORNOT T0199  ; 热压B下层Hip测试气缸上升位延时
OR H0.09  ; 气缸保持（1保持）
ANDLD
OUT 113.08  ; 热压BHip测试气缸上升输出
LD TR0
LD W153.09  ; 热压BHip测试气缸下降[M]
OR W193.09  ; 热压BHip测试气缸下降[A]
OR 113.09  ; 热压BHip测试气缸下降输出
ANDLD
ANDNOT W153.08  ; 热压BHip测试气缸上升[M]
ANDNOT W193.08  ; 热压BHip测试气缸上升[A]
LDNOT T0198  ; 热压B上层Hip测试气缸下降位延时
ORNOT T0200  ; 热压B下层Hip测试气缸下降位延时
OR H0.09  ; 气缸保持（1保持）
ANDLD
OUT 113.09  ; 热压BHip测试气缸下降输出
; rung 26
LD D1001.10  ; 急停（正常=1）
OUT TR0
AND W35.00  ; 4ST_A手动输出允许
AND W113.10  ; 热压B上下层吹气手动
OUT W153.10  ; 热压B上下层吹气[M]
LD TR0
AND W35.01  ; 4ST_A自动输出允许
AND P_Off
OUT W193.10  ; 热压B上下层吹气[A]
LD TR0
LD W153.10  ; 热压B上下层吹气[M]
OR W193.10  ; 热压B上下层吹气[A]
ANDLD
OUT 113.10  ; 热压B上下层吹气输出

